(* CoDeSys 2.3 export: CANOPEN_UNIVERSAL_MASTER.EXP *)
(* Libraries: 05_Utilities\MPLCUtilities.lib 30.1.17 00:00:00, 11_System\SysLibFileAsync.lib 27.1.17 13:50:06, 11_System\SysLibRtc.lib 27.1.17 13:50:06, 12_Additional\Util.lib 27.1.17 13:50:06 *)

(* POU CodeSamples/CANopen/UniversalMaster/PRG_CANopen_IVO_AbsEncoder, FBD *)
(************************************************************************************
*
*                 Code sample  " PRG_CANopen_IVO_AbsEncoder "                 
*
*************************************************************************************
*
* (c) 2009 by SEW-EURODRIVE GmbH & Co KG
*
************************************************************************************
************************************************************************************
*
* PRG_CANopen_IVO_AbsEncoder
*
* This code sample demonstrates, how to configure and connect a 
* CANOpen IVO absolute encoder via CAN.
*
* Remarks : 
* - Use CANopen devices on a separate CAN and don´t mix it with SEW drives.
* - Set the Baudrate in plc configuration 
* 
************************************************************************************)
PROGRAM PRG_CANopen_IVO_AbsEncoder
VAR
	(* Configuration file IVO abs encoder *)
	fbConfig_IVO: FB_Configuration_CANopenSlave_IVO_AbsEncoder;
	stConfig_IVO: MC_EXTENDEDCONFIG_COSLAVE;
	bConfigDone_IVO: BOOL;

	(* Connect IVO abs encoder *)
	fbConnect_IVO: MPLC_ConnectUniversalSlave_CANopen;
	bReset_IVO: BOOL;
	stDiag_IVO: MC_DIAG_COSLAVE;
	aInputs_IVO: ARRAY [1..32] OF ARRAY [1..4] OF WORD;
	aOutputs_IVO: ARRAY [1..32] OF ARRAY [1..4] OF WORD;
	bConnectDone_IVO: BOOL;
	bConnectError_IVO: BOOL;
	nConnectErrorID_IVO: UDINT;
	stAxis_IVO: AXIS_REF;
END_VAR
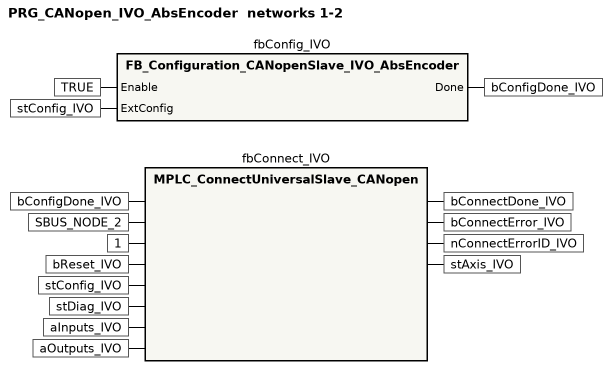
_FBD_ (* Function Block Diagram *)
NETWORK 1
	fbConfig_IVO:FB_Configuration_CANopenSlave_IVO_AbsEncoder(Enable: TRUE, ExtConfig: stConfig_IVO) => bConfigDone_IVO
NETWORK 2
	fbConnect_IVO:MPLC_ConnectUniversalSlave_CANopen(bConfigDone_IVO, SBUS_NODE_2, 1, bReset_IVO, stConfig_IVO, stDiag_IVO, aInputs_IVO, aOutputs_IVO, out 2 => bConnectError_IVO, out 3 => nConnectErrorID_IVO, out 4 => stAxis_IVO) => bConnectDone_IVO
_END_FBD_
(* the same logic as Structured Text *)
(* Network 1 *)
fbConfig_IVO(Enable := TRUE, ExtConfig := stConfig_IVO);
bConfigDone_IVO := fbConfig_IVO.Done;
(* Network 2: see the listing above *)
END_PROGRAM

(* POU CodeSamples/CANopen/UniversalMaster/FB_Configuration_CANopenSlave_IVO_AbsEncoder, ST *)
FUNCTION_BLOCK FB_Configuration_CANopenSlave_IVO_AbsEncoder
VAR_INPUT
	Enable: BOOL; 			(* Activate config *)
END_VAR
VAR_OUTPUT
	Done: BOOL;				(* Config done *)
END_VAR
VAR_IN_OUT
	ExtConfig : MC_EXTENDEDCONFIG_COSLAVE	;
	(*
		########################################################################################################
			MC_EXTENDEDCONFIG_COSLAVE
		#########################################################################################################

						
		Variable								Value			Description
		-------------------------------------------------------------------------------------------------------------------------------------------------------------
		bWaitBeforeOperational 				BOOL;			When TRUE, after the coupler has been parameterized, it won't be switched in operational
																before this variable is FALSE. This can be used for example, to store the configuration with the FB
																MPLC_Universal_CANopen, with Service "SEWIOS_STORE", after a reset of the coppler 
		-------------------------------------------------------------------------------------------------------------------------------------------------------------
		bNoSettingsDownload 				BOOL;			TRUE : No configuration of the module. The configuration has to be done manually.
		-------------------------------------------------------------------------------------------------------------------------------------------------------------
		bResetUnconditional 					BOOL;			Even if the Connect FB isn't in fault it is possible to reset the bus coppler
		-------------------------------------------------------------------------------------------------------------------------------------------------------------
		bIOHold 								BOOL;			TRUE : Input data remain unchanged and the output data are not resetet also if the FB is in fault 
		-------------------------------------------------------------------------------------------------------------------------------------------------------------
		TimeOutHeartBeat					UINT;			If this value (ms) is different to zero, HeartbeatMode will be activated
		-------------------------------------------------------------------------------------------------------------------------------------------------------------
		TimeOutNodeGuarding 				UINT;			If this value (ms) is different to zero, NodeGuarding will be activated. 
																Caution ! The MOVI-PLC basic doesn´t support NodeGuarding 
		-------------------------------------------------------------------------------------------------------------------------------------------------------------
		TimeOutInitSequence					UINT;			Timeout for initialisation sequence (seconds) 
		-------------------------------------------------------------------------------------------------------------------------------------------------------------
		NumberOfRxPDO 					UINT;			Receive PDO : MOVI-PLC --> Slave  max. 32 
		-------------------------------------------------------------------------------------------------------------------------------------------------------------
		NumberOfTxPDO 						UINT;			Send PDO :      Slave --> MOVI-PLC  max 32 
		-------------------------------------------------------------------------------------------------------------------------------------------------------------	
		SyncTime 								USINT;			Cycle time of the sync telegram in ms. 
																Default = 0 : no sync will be started.
																If  SyncTime > 0, this FB initializes a sync telegram with the ID set at SyncCOBID. 
																The slave has to support synchronous communication 
		-------------------------------------------------------------------------------------------------------------------------------------------------------------
		SyncCOBID							UINT;			Index 1005h. ID of the sync telegram. Usually 16#80. IF 0, the ID won't be written.
		-------------------------------------------------------------------------------------------------------------------------------------------------------------
		SyncTimeOut 							INT := -1;		Index 1006h. Normally equal to SyncTime. 
																The slave usually set SyncTimeOut equal to SyncTime * 1.5. 
																If < 0, the index won't be written. 0 means no control over the sync interval 
		-------------------------------------------------------------------------------------------------------------------------------------------------------------
		stInitialParameter_COSlave 			MC_INITIALPARAMETER_COSLAVE;
												(*#################################################################
												With this struct, user defined parameters will be written to the BusCoupler after the
												initialization of the MPLC_ConnectUniversalSlave_CANopen. 
												Add the following code to your program to initialise the struct : 
												Example:
												Index 16#6423:	Activates the event-driven transmission of PDOs with analog inputs
												Index 16#3500:	Index from the manufacturer specific profile area
	
													stInitialParameter_COSlave.aIndex[1] := 16#6423;  	(* Index to write to *)
													stInitialParameter_COSlave.aSubIndex[1] := 0;   	(* SubIndex to write to *)
													stInitialParameter_COSlave.aBytes[1] := 1;   		(* Number of bytes to write  *)
													stInitialParameter_COSlave.aData[1] := 1;   			(* Data *)
	
													stInitialParameter_COSlave.aIndex[2] := 16#3500;  	(* Index to write to *)
													stInitialParameter_COSlave.aSubIndex[2] := 0;   	(* SubIndex to write to *)
													stInitialParameter_COSlave.aBytes[2] := 2;   		(* Number of bytes to write *)
													stInitialParameter_COSlave.aData[2] := 5;   			(* Data *)
	
												If there are more than 10 (DHP11B) or 64 (DHx41B) parameters to write, declare 
												NUMOF_INITIALPARAMETER in your program.
	
													VAR_GLOBAL CONSTANT
														NUMOF_INITIALPARAMETER : UDINT := 20;	
													END_VAR
	
												##################################################################*)
			-------------------------------------------------------------------------------------------------------------------------------------------------------------
		(* IDs of the PDO telegrams. The IDs are always calculated with the following IDs as a basis + the address of the bus coupler *)

		RxPDO 								ARRAY[1..32] OF MC_PDO_COSLAVE;			(* MOVI-PLC --> Slave *)
												(* := 16#200,16#300,16#400,16#500,16#780,16#240,16#340,16#440,16#540,16#7C0;	*)
		-------------------------------------------------------------------------------------------------------------------------------------------------------------
		TxPDO 								ARRAY[1..32] OF MC_PDO_COSLAVE; 			(* Slave --> MOVI-PLC *)
												(*:= 16#180,16#280,16#380,16#480,16#680,16#1C0,16#2C0,16#3C0,16#4C0,16#6C0;*)
	*)
END_VAR
IF Enable AND NOT Done THEN

	(*########################################################

		Configuration of CANopenSlave (IVO AbsEncoder)
		
	#########################################################

		TransmissionType for TxPDOs and RxPDOs:

			0:										Event controlled and sychron (with SYNC-Object)
			1-240:									Cyclic and synchron (with SYNC-Object)
			254:									Producer specified
			255:									Acyclic and eventcontrolled 
			255 and EventTime = InhibitTime:	Cyclic

	#########################################################	*)


	(*************************************************** TxPDOs of CANOpenSlave ( MOVI-PLC ReceiveObjects) ***********************************************************)

	ExtConfig.NumberOfTxPDO				:= 1;		(*  TxPDO ---> CANopenSlave Transmit *)

	ExtConfig.TxPDO[1].EventTime			:= 20;		(* Slave: Index 0x18xx SubIndex 5: CycleTime in ms for CANopenSlave TXPDO *)
	ExtConfig.TxPDO[1].InhibitTime			:= 20;		(* Slave: Index 0x18xx SubIndex 3: InhibitTime in ms for CANopenSlave TxPDO *)
	ExtConfig.TxPDO[1].TransmissionType	:= 254;		(* Slave: Index 0x18xx SubIndex 2: TransmissionType for this TxPDO *)


	(*************************************************** RxPDOs of CANOpenSlave ( MOVI-PLC TransmitObjects) **********************************************************)

	ExtConfig.NumberOfRxPDO				:= 0;		(*  RxPDO ---> CANopenSlave Receive *)

	(* ExtConfig.RxPDO[1].EventTime		:= 0;		(* Master: CycleTime in ms for TransmitObjects (MOVI-PLC) *)
	ExtConfig.RxPDO[1].InhibitTime			:= 0;		(* Master: InhibitTime in ms for TransmitObjects (MOVI-PLC) *)
	ExtConfig.RxPDO[1].Length				:= 2;		(* Master: Length of this TransmitObject in bytes *)
	ExtConfig.RxPDO[1].TransmissionType	:= 255;		(* Slave: Index 0x14xx SubIndex 2: TransmissionType for this RxPDO *)*)


	(***************************************************** Additional parameters to set in the CANOpenSlave  ***************************************************************)

	(* Set rotation direction *)
	ExtConfig.stInitialParameter_COSlave.aIndex[1]			:= 16#6000;
	ExtConfig.stInitialParameter_COSlave.aSubIndex[1]	:= 0;
	ExtConfig.stInitialParameter_COSlave.aBytes[1]		:= 2;
	ExtConfig.stInitialParameter_COSlave.aData[1]			:= 0;		(* 0 = CV, 1 = CCV *)

	(* Write reference offset to AbsEncoder, Index 6003.0, data = new position *)
	(* Write Delivery state to AbsEncoder, Index 1011.1, data = 16#6C_6F_61_64 (load) *)
	(* Save values in Flash memory in the AbsEncoder, Index 1010.1, data = 16#73_61_76_65 (save) *)


	(********************************************** Additional configuration. Default values are in most cases sufficient *****************************************************)

	ExtConfig.bIOHold						:= FALSE;
	ExtConfig.bNoSettingsDownload			:= FALSE;
	ExtConfig.bWaitBeforeOperational		:= FALSE;
	ExtConfig.bResetUnconditional			:= FALSE;

	ExtConfig.TimeOutHeartBeat				:= 400;				(* [ms] *)
	ExtConfig.TimeOutNodeGuarding		:= 0;				(* [ms]. CAUTION ! DHP11B (MOVI-PLC basic) does NOT support NodeGuarding *)
	ExtConfig.TimeOutInitSequence			:= 5;				(* [seconds]. If the Init-Sequence takes longer than this TimeOut time --> Error *)
	ExtConfig.SyncCOBID						:= 0;				(* SyncObject ID for TransmissionType 0-240 (RxPDO). Usually 128. If 0, the ID will not be written *)
	ExtConfig.SyncTime						:= 0;				(* CycleTime for the SYNC-Object *)

	ExtConfig.TxPDO[1].COBID				:= 16#180;			(* In order to disable the use of RTR frames for the PDOs, set bit 30 = "RTR not allowed" *)
	ExtConfig.TxPDO[2].COBID				:= 16#280;			(* Ex. 16#4000_0280 *)
	ExtConfig.TxPDO[3].COBID				:= 16#380;
	ExtConfig.TxPDO[4].COBID				:= 16#480;			(* NOTE! These values are base values. The input "Address" will automatically be added *)
	ExtConfig.TxPDO[5].COBID				:= 16#680;
	ExtConfig.TxPDO[6].COBID				:= 16#1C0;
	ExtConfig.TxPDO[7].COBID				:= 16#2C0;
	ExtConfig.TxPDO[8].COBID				:= 16#3C0;
	ExtConfig.TxPDO[9].COBID				:= 16#4C0;
	ExtConfig.TxPDO[10].COBID				:= 16#6C0;

	ExtConfig.RxPDO[1].COBID				:= 16#200;
	ExtConfig.RxPDO[2].COBID				:= 16#300;
	ExtConfig.RxPDO[3].COBID				:= 16#400;
	ExtConfig.RxPDO[4].COBID				:= 16#500;
	ExtConfig.RxPDO[5].COBID				:= 16#780;
	ExtConfig.RxPDO[6].COBID				:= 16#240;
	ExtConfig.RxPDO[7].COBID				:= 16#340;
	ExtConfig.RxPDO[8].COBID				:= 16#440;
	ExtConfig.RxPDO[9].COBID				:= 16#540;
	ExtConfig.RxPDO[10].COBID				:= 16#7C0;

	Done := TRUE;

END_IF
END_FUNCTION_BLOCK

(* POU CodeSamples/CANopen/UniversalMaster/CANopen_activ, ST *)
(*######################################################
Functionblock:
- to send sync for the slave, to auto-detection of baudrate.
- set baudrate 
- set address 
#######################################################*)
FUNCTION_BLOCK CANopen_activ
VAR_INPUT
	Node: CAN_NODE; (* CAN_NODE_1 or CAN_NODE_2*)
	Address_Default : WORD;(* 0...127*)
	Address: WORD;			(* 1...63 *)
	Baudrate: WORD;(* 0 = 1 M , 2 = 500 k , 3 = 250 k baud*)
END_VAR
VAR_OUTPUT
	Done: BOOL; 				(* Connection to the CAN module successfully started *)
	Error: BOOL; 				(* Error within the function block *)
	ErrorID: UDINT; 			(* Error identification *)
END_VAR
VAR
	Init: BOOL;
	CanMsg: ST_CanAcyclicMsg;
	Timer: TON;
	l_State: UINT;
	StartAdresse_Diag: UINT;
	StartAdresse_Input: UINT;
	StartAdresse_Output: UINT;
	bMerkerCANSuspended: BOOL;
	SComCtrl1: SComControl;
	Counter: INT;
	fbSComCheckId: SComCheckId;
	SComRecSDO: SComReceive;
	SComRecNMT: SComReceive;
	SComRecEmergency: SComReceive;
	sSDORecDataTemp : sTwoDWORDData;
	NMT_Default_Byte : BYTE;
	NMT_Byte : BYTE;
	AbortCode: DWORD;
END_VAR
CASE l_State OF
(* ============ Initialisierung  Variablen =============== *)
	0:
		l_State := 10;

	10:
		IF ( Address < 1 ) OR ( Address > 63 ) OR (Address_Default > 127) THEN
			Error := TRUE;
			ErrorID := E_CAN_IO_MODULE_INVALID_PARAMETERS;
			RETURN;
		END_IF

		l_State := 50;

	50:
	(* SBus suspend --> damit können neue Objekte eingerichtet werden*)
      (* SCOM SUSPEND *)
	IF fTestAndSet( stInterlock.yTaskLock_CANSuspend ) THEN		(* CAN "belegen" damit keine andere Instanz Objekte anlegen will *)
		SEWMotionIntern.SComAllocationMax_I := SEWMotionIntern.SComAllocationMax_I - ( 12 + 4 * 2(*( xx.NbTxPDO + xx.NbCyclicRxPDO )*));
		SEWMotionIntern.SComAllocationMax_M := SEWMotionIntern.SComAllocationMax_M - ( 12 + 4 *2(* ( xx.NbTxPDO + xx.NbCyclicRxPDO )*));
		SEWMotionIntern.SComAllocationMax_Q := SEWMotionIntern.SComAllocationMax_Q - ( 12 + 4 * 2(*( xx.NbTxPDO + xx.NbCyclicRxPDO )*));
		StartAdresse_Diag := DWORD_TO_UINT (SEWMotionIntern.SComAllocationMax_M );
		StartAdresse_Input := DWORD_TO_UINT( SEWMotionIntern.SComAllocationMax_I );
		StartAdresse_Output := DWORD_TO_UINT( SEWMotionIntern.SComAllocationMax_Q );
		bMerkerCANSuspended := TRUE;
		SComCtrl1( Execute := FALSE );
		l_State := 60;
	END_IF

	60:
	(* SBus suspend --> damit können neue Objekte eingerichtet werden*)
      (* SCOM SUSPEND *)
	SComCtrl1(
		Execute := TRUE,
		Node := Node,
	 	Control := SCOM_CONTROL_SUSPEND,
		Error => Error,
		ErrorID => ErrorID );
       IF SComCtrl1.Done THEN
		l_State := 65;
	END_IF

	65:
	(* ID´s überprüfen für Adresse Default --> könnte durch andere SCOM Objekte schon belegt sein *)
	FOR Counter := 1 TO 6 DO
		IF (Counter = 6 )  THEN
			fbSComCheckId(
				Enable := TRUE,
				Node := Node,
				Id := 16#80);
		ELSE
			fbSComCheckId(
				Enable := TRUE,
				Node := Node,
				Id := ( Address_Default + aCOB_IDs_general_CO[Counter] ));
		END_IF
		IF fbSComCheckId.IsUsed OR NOT fbSComCheckId.Done OR ((Counter < 6 ) AND ( fbSComCheckId.Id = 16#80)) THEN
			Error := TRUE;
			ErrorID := E_CAN_IO_MODULE_CAN_ID_ERROR ;
			RETURN;
		ELSIF fbSComCheckId.Error THEN
			Error := TRUE;
			ErrorID := fbSComCheckId.ErrorID;
			RETURN;
		END_IF
	END_FOR
	l_State := 66;

	66:
	(* ID´s überprüfen für Adresse  --> könnte durch andere SCOM Objekte schon belegt sein *)
	FOR Counter := 1 TO 6 DO
		IF (Counter = 6 )  THEN
			fbSComCheckId(
				Enable := TRUE,
				Node := Node,
				Id := 16#80);
		ELSE
			fbSComCheckId(
				Enable := TRUE,
				Node := Node,
				Id := ( Address + aCOB_IDs_general_CO[Counter] ));
		END_IF
		IF fbSComCheckId.IsUsed OR NOT fbSComCheckId.Done OR ((Counter < 6 ) AND ( fbSComCheckId.Id = 16#80)) THEN
			Error := TRUE;
			ErrorID := E_CAN_IO_MODULE_CAN_ID_ERROR ;
			RETURN;
		ELSIF fbSComCheckId.Error THEN
			Error := TRUE;
			ErrorID := fbSComCheckId.ErrorID;
			RETURN;
		END_IF
	END_FOR
	SComRecSDO( Execute := FALSE );
	l_State := 70;

	70:
	(* Receive Objekt für Antwort Hochlauf Address_Default anlegen SDO*)
	SComRecSDO(
		Execute := TRUE,
		Node := Node,
		ID := 16#580 + Address_Default,
		Length := 8,
		DataDest := StartAdresse_Input,
		DiagDest := StartAdresse_Diag,
		Error => Error,
		ErrorID => ErrorID );
	IF SComRecSDO.Done THEN
		StartAdresse_Input := StartAdresse_Input + 4;
		StartAdresse_Diag := StartAdresse_Diag + 4;
		StartAdresse_Output := StartAdresse_Output + 4;
		SEWInternCOSlave[Address_Default].LibIn := SComRecSDO.DataDest;
		SComRecNMT( Execute := FALSE );
   		 l_State := 72;
	END_IF

	72:
	(* Receive Objekt für Antwort Hochlauf Address_Default anlegen NMT*)
	SComRecNMT(
		Execute := TRUE,
		Node := Node,
		ID := 16#700 + Address_Default,
		Length := 1,
		DataDest := StartAdresse_Input,
		DiagDest := StartAdresse_Diag,
		Error => Error,
		ErrorID => ErrorID );
	IF SComRecSDO.Done THEN
		StartAdresse_Input := StartAdresse_Input + 2;
		StartAdresse_Diag := StartAdresse_Diag + 2;
		StartAdresse_Output := StartAdresse_Output + 2;
		SComRecNMT( Execute := FALSE );
   		 l_State := 73;
	END_IF

	73:
	(* Receive Objekt für Antwort Hochlauf Address anlegen NMT*)
	SComRecNMT(
		Execute := TRUE,
		Node := Node,
		ID := 16#700 + Address,
		Length := 8,
		DataDest := StartAdresse_Input,
		DiagDest := StartAdresse_Diag,
		Error => Error,
		ErrorID => ErrorID );
	IF SComRecSDO.Done THEN
		StartAdresse_Input := StartAdresse_Input + 2;
		StartAdresse_Diag := StartAdresse_Diag + 2;
		StartAdresse_Output := StartAdresse_Output + 2;
		SComRecEmergency( Execute := FALSE );
   		 l_State := 74;
	END_IF

	74:
	(* Receive Objekt für Emergency Object einstellen *)
   	 SComRecEmergency(
		Execute := TRUE,
		Node := Node,
		ID := 16#80 + Address_Default,
		Length := 8,
		DataDest := StartAdresse_Input,
		DiagDest := StartAdresse_Diag,
		Error => Error,
		ErrorID => ErrorID);
	IF SComRecEmergency.Done THEN
		SComCtrl1( Execute := FALSE );
		l_State := 80;
	END_IF

	80:
	(* SBUS einschalten *)
	SComCtrl1(
		Execute := TRUE,
		Node := Node,
		Control := SCOM_CONTROL_ON );
	(* SBUS Initialisierung abgeschlossen *)
	IF SComCtrl1.Done THEN
		stInterlock.yTaskLock_CANSuspend := 0;
		bMerkerCANSuspended := FALSE;
		l_State := 90;
	END_IF

	90:
	(* Synch senden damit der Slave die Baudrate erkennt *)
		IF NOT Init THEN
			CanMsg := F_WriteCanMsg(
										Node := Node,
										ID := 16#80,
										Length := 1,
										Data1:= 0,
										Data2 := 0,
										Data3 := 0,
										Data4 := 0,
										SBUSGateway_LogAdr := 0 );
			IF ( CanMsg.State = GEN_1_BUFFSTATE_INSERTED ) THEN
				Init :=TRUE;
			END_IF
		ELSIF Init THEN
			CanMsg.Result :=F_ResultCanMsg(CanAcyclicMsg := CanMsg);
			IF ( CanMsg.Result = GEN_3_BUFFSTATE_COMPLETED_SUCCESSFUL ) THEN
				Init := FALSE;
				l_State := 92;
			(* Fehler beim Senden --> Nachricht ging verloren --> nochmals *)
			ELSIF (CanMsg.Result = GEN_5_BUFFSTATE_COMPLETED_MSG_LOST ) THEN
				Init := FALSE;
			(* Fehler beim Senden --> Non-recovery error from CAN --> nochmals *)
			ELSIF (CanMsg.Result = GEN_4_BUFFSTATE_COMPLETED_ERROR ) THEN
				Init := FALSE;
			END_IF
		END_IF

	92: (* Kontrolle ob Slave mit Address_Default antwortet *)
	Timer(	IN := TRUE, PT := t#1s );
	IF NOT Timer.Q THEN
		ConfDataEx_ReadFromIoBuffer( SEWInternCOSlave[Address_Default].LibIn+4, BUFSEL_IN, ADR(NMT_Default_Byte), 1);
		ConfDataEx_ReadFromIoBuffer( SEWInternCOSlave[Address_Default].LibIn+6, BUFSEL_IN, ADR(NMT_Byte), 1);
		IF NMT_Default_Byte = 0 THEN
			IF NMT_Byte = 0 THEN
				l_State := 90;
			ELSE
				l_State := 100;
			END_IF
		ELSE
			l_State := 100;
		END_IF
	ELSE
		l_State := 100;
	END_IF

	100:
	(* Baudrate einstellen *)
	Timer(	IN := TRUE, PT := t#100ms );
	IF Timer.Q THEN
		IF NOT Init THEN
			CanMsg := F_WriteCanMsg(
										Node := Node,
										ID := 16#600+Address_Default,
										Length := 8,
										Data1:= 16#2F00,
										Data2 := 16#2100,
										Data3 := SHL(Baudrate,8),
										Data4 := 0,
										SBUSGateway_LogAdr := 0 );
			IF ( CanMsg.State = GEN_1_BUFFSTATE_INSERTED ) THEN
				Init :=TRUE;
			END_IF
		ELSIF Init THEN
			CanMsg.Result :=F_ResultCanMsg(CanAcyclicMsg := CanMsg);
			IF ( CanMsg.Result = GEN_3_BUFFSTATE_COMPLETED_SUCCESSFUL ) THEN
				Init := FALSE;
				Timer( IN := FALSE );
				l_State := 110;
			(* Fehler beim Senden --> Nachricht ging verloren --> nochmals *)
			ELSIF (CanMsg.Result = GEN_5_BUFFSTATE_COMPLETED_MSG_LOST ) THEN
				Init := FALSE;
				Timer( IN := FALSE );
			(* Fehler beim Senden --> Non-recovery error from CAN --> nochmals *)
			ELSIF (CanMsg.Result = GEN_4_BUFFSTATE_COMPLETED_ERROR ) THEN
				Init := FALSE;
				Timer( IN := FALSE );
			END_IF
		END_IF
	END_IF

	110:
		ConfDataEx_ReadFromIoBuffer( SEWInternCOSlave[Address_Default].LibIn, BUFSEL_IN, ADR(sSDORecDataTemp), 8);
		IF MAX_NUMBER_AXIS <> 12 THEN
			sSDORecDataTemp.DWORD1 := fSwapUDINTtoIntel(sSDORecDataTemp.DWORD1);
			sSDORecDataTemp.DWORD2 := fSwapUDINTtoIntel(sSDORecDataTemp.DWORD2);
		END_IF
		IF (sSDORecDataTemp.DWORD1 AND 16#FFFF_FFF0) = (16#0021002F AND 16#FFFF_FF00) + 16#60 THEN
				l_State := 120;
		ELSIF sSDORecDataTemp.DWORD1= (16#0021002F AND 16#FFFF_FF00) + 16#80 THEN
			Error := TRUE;
			ErrorID := E_CAN_IO_MODULE_INVALID_PARAMETERS;			(* Parameter error *)
			AbortCode := sSDORecDataTemp.DWORD2;	(* SDO abort code *)
		ELSE
			(* Time out *)
			Timer( IN := TRUE, PT := T#500ms);
			IF Timer.Q THEN
				Error := TRUE;
				ErrorID := E_CAN_IO_MODULE_TIME_OUT_SBUS;			(* Parameter transfer Time out *)
			END_IF
		END_IF

	120:
	(* ID einstellen *)
	Timer(	IN := TRUE, PT := t#100ms );
	IF Timer.Q THEN
		IF NOT Init THEN
			CanMsg := F_WriteCanMsg(
										Node := Node,
										ID := 16#600+Address_Default,
										Length := 8,
										Data1:= 16#2F01,
										Data2 := 16#2100,
										Data3 := SHL(Address,8),
										Data4 := 0,
										SBUSGateway_LogAdr := 0 );
			IF ( CanMsg.State = GEN_1_BUFFSTATE_INSERTED ) THEN
				Init :=TRUE;
			END_IF
		ELSIF Init THEN
			CanMsg.Result :=F_ResultCanMsg(CanAcyclicMsg := CanMsg);
			IF ( CanMsg.Result = GEN_3_BUFFSTATE_COMPLETED_SUCCESSFUL ) THEN
				Init := FALSE;
				Timer( IN := FALSE );
				l_State := 130;
			(* Fehler beim Senden --> Nachricht ging verloren --> nochmals *)
			ELSIF (CanMsg.Result = GEN_5_BUFFSTATE_COMPLETED_MSG_LOST ) THEN
				Init := FALSE;
				Timer( IN := FALSE );
			(* Fehler beim Senden --> Non-recovery error from CAN --> nochmals *)
			ELSIF (CanMsg.Result = GEN_4_BUFFSTATE_COMPLETED_ERROR ) THEN
				Init := FALSE;
				Timer( IN := FALSE );
			END_IF
		END_IF
	END_IF

	130:
		ConfDataEx_ReadFromIoBuffer( SEWInternCOSlave[Address_Default].LibIn, BUFSEL_IN, ADR(sSDORecDataTemp), 8);
		IF MAX_NUMBER_AXIS <> 12 THEN
			sSDORecDataTemp.DWORD1 := fSwapUDINTtoIntel(sSDORecDataTemp.DWORD1);
			sSDORecDataTemp.DWORD2 := fSwapUDINTtoIntel(sSDORecDataTemp.DWORD2);
		END_IF
		IF (sSDORecDataTemp.DWORD1 AND 16#FFFF_FFF0) = (16#0021012F AND 16#FFFF_FF00) + 16#60 THEN
				l_State := 140;
		ELSIF sSDORecDataTemp.DWORD1= (16#0021012F AND 16#FFFF_FF00) + 16#80 THEN
			Error := TRUE;
			ErrorID := E_CAN_IO_MODULE_INVALID_PARAMETERS;			(* Parameter error *)
			AbortCode := sSDORecDataTemp.DWORD2;	(* SDO abort code *)
		ELSE
			(* Time out *)
			Timer( IN := TRUE, PT := T#500ms);
			IF Timer.Q THEN
				Error := TRUE;
				ErrorID := E_CAN_IO_MODULE_TIME_OUT_SBUS;			(* Parameter transfer Time out *)
			END_IF
		END_IF

	140:
	(* Parameter save *)
	Timer(	IN := TRUE, PT := t#100ms );
	IF Timer.Q THEN
		IF NOT Init THEN
			CanMsg := F_WriteCanMsg(
										Node := Node,
										ID := 16#600+Address_Default,
										Length := 8,
										Data1:= 16#2310,
										Data2 := 16#1001,
										Data3 := 16#7361,
										Data4 := 16#7665,
										SBUSGateway_LogAdr := 0 );
			IF ( CanMsg.State = GEN_1_BUFFSTATE_INSERTED ) THEN
				Init :=TRUE;
			END_IF
		ELSIF Init THEN
			CanMsg.Result :=F_ResultCanMsg(CanAcyclicMsg := CanMsg);
			IF ( CanMsg.Result = GEN_3_BUFFSTATE_COMPLETED_SUCCESSFUL ) THEN
				Init := FALSE;
				Timer( IN := FALSE );
				l_State := 150;
			(* Fehler beim Senden --> Nachricht ging verloren --> nochmals *)
			ELSIF (CanMsg.Result = GEN_5_BUFFSTATE_COMPLETED_MSG_LOST ) THEN
				Init := FALSE;
				Timer( IN := FALSE );
			(* Fehler beim Senden --> Non-recovery error from CAN --> nochmals *)
			ELSIF (CanMsg.Result = GEN_4_BUFFSTATE_COMPLETED_ERROR ) THEN
				Init := FALSE;
				Timer( IN := FALSE );
			END_IF
		END_IF
	END_IF

	150:
		ConfDataEx_ReadFromIoBuffer( SEWInternCOSlave[Address_Default].LibIn, BUFSEL_IN, ADR(sSDORecDataTemp), 8);
		IF MAX_NUMBER_AXIS <> 12 THEN
			sSDORecDataTemp.DWORD1 := fSwapUDINTtoIntel(sSDORecDataTemp.DWORD1);
			sSDORecDataTemp.DWORD2 := fSwapUDINTtoIntel(sSDORecDataTemp.DWORD2);
		END_IF
		IF (sSDORecDataTemp.DWORD1 AND 16#FFFF_FFF0) = (16#01101023 AND 16#FFFF_FF00) + 16#60 THEN
				l_State := 200;
		ELSIF sSDORecDataTemp.DWORD1= (16#01101023 AND 16#FFFF_FF00) + 16#80 THEN
			Error := TRUE;
			ErrorID := E_CAN_IO_MODULE_INVALID_PARAMETERS;			(* Parameter error *)
			AbortCode := sSDORecDataTemp.DWORD2;	(* SDO abort code *)
		ELSE
			(* Time out *)
			Timer( IN := TRUE, PT := T#500ms);
			IF Timer.Q THEN
				Error := TRUE;
				ErrorID := E_CAN_IO_MODULE_TIME_OUT_SBUS;			(* Parameter transfer Time out *)
			END_IF
		END_IF

	200:
		Done := TRUE;
		Error := FALSE;
		ErrorID := 0;

END_CASE
END_FUNCTION_BLOCK

(* POU CodeSamples/CANopen/UniversalMaster/FB_Configuration_CANopenSlave_Beckhoff_BK5120, ST *)
FUNCTION_BLOCK FB_Configuration_CANopenSlave_Beckhoff_BK5120
VAR_INPUT
	Enable: BOOL; 			(* Activate config *)
END_VAR
VAR_OUTPUT
	Done: BOOL;				(* Config done *)
END_VAR
VAR_IN_OUT
	ExtConfig : MC_EXTENDEDCONFIG_COSLAVE	;
	(*
		########################################################################################################
			MC_EXTENDEDCONFIG_COSLAVE
		#########################################################################################################

						
		Variable								Value			Description
		-------------------------------------------------------------------------------------------------------------------------------------------------------------
		bWaitBeforeOperational 				BOOL;			When TRUE, after the coupler has been parameterized, it won't be switched in operational
																before this variable is FALSE. This can be used for example, to store the configuration with the FB
																MPLC_Universal_CANopen, with Service "SEWIOS_STORE", after a reset of the coppler 
		-------------------------------------------------------------------------------------------------------------------------------------------------------------
		bNoSettingsDownload 				BOOL;			TRUE : No configuration of the module. The configuration has to be done manually.
		-------------------------------------------------------------------------------------------------------------------------------------------------------------
		bResetUnconditional 					BOOL;			Even if the Connect FB isn't in fault it is possible to reset the bus coppler
		-------------------------------------------------------------------------------------------------------------------------------------------------------------
		bIOHold 								BOOL;			TRUE : Input data remain unchanged and the output data are not resetet also if the FB is in fault 
		-------------------------------------------------------------------------------------------------------------------------------------------------------------
		TimeOutHeartBeat					UINT;			If this value (ms) is different to zero, HeartbeatMode will be activated
		-------------------------------------------------------------------------------------------------------------------------------------------------------------
		TimeOutNodeGuarding 				UINT;			If this value (ms) is different to zero, NodeGuarding will be activated. 
																Caution ! The MOVI-PLC basic doesn´t support NodeGuarding 
		-------------------------------------------------------------------------------------------------------------------------------------------------------------
		TimeOutInitSequence					UINT;			Timeout for initialisation sequence (seconds) 
		-------------------------------------------------------------------------------------------------------------------------------------------------------------
		NumberOfRxPDO 					UINT;			Receive PDO : MOVI-PLC --> Slave  max. 32 
		-------------------------------------------------------------------------------------------------------------------------------------------------------------
		NumberOfTxPDO 						UINT;			Send PDO :      Slave --> MOVI-PLC  max 32 
		-------------------------------------------------------------------------------------------------------------------------------------------------------------	
		SyncTime 								USINT;			Cycle time of the sync telegram in ms. 
																Default = 0 : no sync will be started.
																If  SyncTime > 0, this FB initializes a sync telegram with the ID set at SyncCOBID. 
																The slave has to support synchronous communication 
		-------------------------------------------------------------------------------------------------------------------------------------------------------------
		SyncCOBID							UINT;			Index 1005h. ID of the sync telegram. Usually 16#80. IF 0, the ID won't be written.
		-------------------------------------------------------------------------------------------------------------------------------------------------------------
		SyncTimeOut 							INT := -1;		Index 1006h. Normally equal to SyncTime. 
																The slave usually set SyncTimeOut equal to SyncTime * 1.5. 
																If < 0, the index won't be written. 0 means no control over the sync interval 
		-------------------------------------------------------------------------------------------------------------------------------------------------------------
		stInitialParameter_COSlave 			MC_INITIALPARAMETER_COSLAVE;
												(*#################################################################
												With this struct, user defined parameters will be written to the BusCoupler after the
												initialization of the MPLC_ConnectUniversalSlave_CANopen. 
												Add the following code to your program to initialise the struct : 
												Example:
												Index 16#6423:	Activates the event-driven transmission of PDOs with analog inputs
												Index 16#3500:	Index from the manufacturer specific profile area
	
													stInitialParameter_COSlave.aIndex[1] := 16#6423;  	(* Index to write to *)
													stInitialParameter_COSlave.aSubIndex[1] := 0;   	(* SubIndex to write to *)
													stInitialParameter_COSlave.aBytes[1] := 1;   		(* Number of bytes to write  *)
													stInitialParameter_COSlave.aData[1] := 1;   			(* Data *)
	
													stInitialParameter_COSlave.aIndex[2] := 16#3500;  	(* Index to write to *)
													stInitialParameter_COSlave.aSubIndex[2] := 0;   	(* SubIndex to write to *)
													stInitialParameter_COSlave.aBytes[2] := 2;   		(* Number of bytes to write *)
													stInitialParameter_COSlave.aData[2] := 5;   			(* Data *)
	
												If there are more than 10 (DHP11B) or 64 (DHx41B) parameters to write, declare 
												NUMOF_INITIALPARAMETER in your program.
	
													VAR_GLOBAL CONSTANT
														NUMOF_INITIALPARAMETER : UDINT := 20;	
													END_VAR
	
												##################################################################*)
			-------------------------------------------------------------------------------------------------------------------------------------------------------------
		(* IDs of the PDO telegrams. The IDs are always calculated with the following IDs as a basis + the address of the bus coupler *)

		RxPDO 								ARRAY[1..32] OF MC_PDO_COSLAVE;			(* MOVI-PLC --> Slave *)
												(* := 16#200,16#300,16#400,16#500,16#780,16#240,16#340,16#440,16#540,16#7C0;	*)
		-------------------------------------------------------------------------------------------------------------------------------------------------------------
		TxPDO 								ARRAY[1..32] OF MC_PDO_COSLAVE; 			(* Slave --> MOVI-PLC *)
												(*:= 16#180,16#280,16#380,16#480,16#680,16#1C0,16#2C0,16#3C0,16#4C0,16#6C0;*)
	*)
END_VAR
IF Enable AND NOT Done THEN

	(*########################################################

		Configuration of CANopenSlave (Beckhoff BK5120)
		
	#########################################################

		TransmissionType for TxPDOs and RxPDOs:

			0:										Event controlled and sychron (with SYNC-Object)
			1-240:									Cyclic and synchron (with SYNC-Object)
			254:									Producer specified
			255:									Acyclic and eventcontrolled 
			255 and EventTime = InhibitTime:	Cyclic

	#########################################################	*)


	(*************************************************** TxPDOs of CANOpenSlave ( MOVI-PLC ReceiveObjects) ***********************************************************)

	ExtConfig.NumberOfTxPDO				:= 2;		(*  TxPDO ---> CANopenSlave Transmit *)

	ExtConfig.TxPDO[1].EventTime			:= 200;		(* Slave: Index 0x18xx SubIndex 5: CycleTime in ms for CANopenSlave TXPDO *)
	ExtConfig.TxPDO[1].InhibitTime			:= 5;		(* Slave: Index 0x18xx SubIndex 3: InhibitTime in ms for CANopenSlave TxPDO *)
	ExtConfig.TxPDO[1].TransmissionType	:= 255;		(* Slave: Index 0x18xx SubIndex 2: TransmissionType for this TxPDO *)

	ExtConfig.TxPDO[2].EventTime			:= 100;		(* Slave: Index 0x18xx SubIndex 5: CycleTime in ms for CANopenSlave TXPDO *)
	ExtConfig.TxPDO[2].InhibitTime			:= 100;		(* Slave: Index 0x18xx SubIndex 3: InhibitTime in ms for CANopenSlave TxPDO *)
	ExtConfig.TxPDO[2].TransmissionType	:= 255;		(* Slave: Index 0x18xx SubIndex 2: TransmissionType for this TxPDO *)


	(*************************************************** RxPDOs of CANOpenSlave ( MOVI-PLC TransmitObjects) **********************************************************)

	ExtConfig.NumberOfRxPDO				:= 2;		(*  RxPDO ---> CANopenSlave Receive *)

	ExtConfig.RxPDO[1].EventTime			:= 200;		(* Master: CycleTime in ms for TransmitObjects (MOVI-PLC) *)
	ExtConfig.RxPDO[1].InhibitTime			:= 5;		(* Master: InhibitTime in ms for TransmitObjects (MOVI-PLC) *)
	ExtConfig.RxPDO[1].Length				:= 8;		(* Master: Length of this TransmitObject in bytes *)
	ExtConfig.RxPDO[1].TransmissionType	:= 255;		(* Slave: Index 0x14xx SubIndex 2: TransmissionType for this RxPDO *)

	ExtConfig.RxPDO[2].EventTime			:= 100;		(* Master: CycleTime in ms for TransmitObjects (MOVI-PLC) *)
	ExtConfig.RxPDO[2].InhibitTime			:= 100;		(* Master: InhibitTime in ms for TransmitObjects (MOVI-PLC) *)
	ExtConfig.RxPDO[2].Length				:= 8;		(* Master: Length of this TransmitObject in bytes *)
	ExtConfig.RxPDO[2].TransmissionType	:= 255;		(* Slave: Index 0x14xx SubIndex 2: TransmissionType for this RxPDO *)


	(***************************************************** Additional parameters to set in the CANOpenSlave  ***************************************************************)

	(* Enable transmission of analog inputs *)
	ExtConfig.stInitialParameter_COSlave.aIndex[1]			:= 16#6423;
	ExtConfig.stInitialParameter_COSlave.aSubIndex[1]	:= 0;
	ExtConfig.stInitialParameter_COSlave.aBytes[1]		:= 1;
	ExtConfig.stInitialParameter_COSlave.aData[1]			:= 1;

(*	(* Disable write protection, step 1 *)
	ExtConfig.stInitialParameter_COSlave.aIndex[2]			:= 16#4500;
	ExtConfig.stInitialParameter_COSlave.aSubIndex[2]	:= 0;
	ExtConfig.stInitialParameter_COSlave.aBytes[2]		:= 4;
	ExtConfig.stInitialParameter_COSlave.aData[2]			:= 16#E302_AFFE;

	(* Disable write protection, step 2 *)
	ExtConfig.stInitialParameter_COSlave.aIndex[3]			:= 16#4500;
	ExtConfig.stInitialParameter_COSlave.aSubIndex[3]	:= 0;
	ExtConfig.stInitialParameter_COSlave.aBytes[3]		:= 4;
	ExtConfig.stInitialParameter_COSlave.aData[3]			:= 16#E301_0001;

	(* Disable write protection, step 3 *)
	ExtConfig.stInitialParameter_COSlave.aIndex[4]			:= 16#4500;
	ExtConfig.stInitialParameter_COSlave.aSubIndex[4]	:= 0;
	ExtConfig.stInitialParameter_COSlave.aBytes[4]		:= 4;
	ExtConfig.stInitialParameter_COSlave.aData[4]			:= 16#E300_0101;
*)

	(********************************************** Additional configuration. Default values are in most cases sufficient *****************************************************)

	ExtConfig.bIOHold						:= FALSE;
	ExtConfig.bNoSettingsDownload			:= FALSE;
	ExtConfig.bWaitBeforeOperational		:= FALSE;
	ExtConfig.bResetUnconditional			:= FALSE;

	ExtConfig.TimeOutHeartBeat				:= 400;				(* [ms] *)
	ExtConfig.TimeOutNodeGuarding		:= 0;				(* [ms]. CAUTION ! DHP11B (MOVI-PLC basic) does NOT support NodeGuarding *)
	ExtConfig.TimeOutInitSequence			:= 10;				(* [seconds]. If the Init-Sequence takes longer than this TimeOut time --> Error *)
	ExtConfig.SyncCOBID						:= 0;				(* SyncObject ID for TransmissionType 0-240 (RxPDO). Usually 128. If 0, the ID will not be written *)
	ExtConfig.SyncTime						:= 0;				(* CycleTime for the SYNC-Object *)

	ExtConfig.TxPDO[1].COBID				:= 16#180;			(* In order to disable the use of RTR frames for the PDOs, set bit 30 = "RTR not allowed" *)
	ExtConfig.TxPDO[2].COBID				:= 16#280;			(* Ex. 16#4000_0280 *)
	ExtConfig.TxPDO[3].COBID				:= 16#380;
	ExtConfig.TxPDO[4].COBID				:= 16#480;			(* NOTE! These values are base values. The input "Address" will automatically be added *)
	ExtConfig.TxPDO[5].COBID				:= 16#680;
	ExtConfig.TxPDO[6].COBID				:= 16#1C0;
	ExtConfig.TxPDO[7].COBID				:= 16#2C0;
	ExtConfig.TxPDO[8].COBID				:= 16#3C0;
	ExtConfig.TxPDO[9].COBID				:= 16#4C0;
	ExtConfig.TxPDO[10].COBID				:= 16#6C0;

	ExtConfig.RxPDO[1].COBID				:= 16#200;
	ExtConfig.RxPDO[2].COBID				:= 16#300;
	ExtConfig.RxPDO[3].COBID				:= 16#400;
	ExtConfig.RxPDO[4].COBID				:= 16#500;
	ExtConfig.RxPDO[5].COBID				:= 16#780;
	ExtConfig.RxPDO[6].COBID				:= 16#240;
	ExtConfig.RxPDO[7].COBID				:= 16#340;
	ExtConfig.RxPDO[8].COBID				:= 16#440;
	ExtConfig.RxPDO[9].COBID				:= 16#540;
	ExtConfig.RxPDO[10].COBID				:= 16#7C0;

	Done := TRUE;

END_IF
END_FUNCTION_BLOCK

(* POU CodeSamples/CANopen/UniversalMaster/FB_Configuration_CANopenSlave_FESTO_CPX, ST *)
FUNCTION_BLOCK FB_Configuration_CANopenSlave_FESTO_CPX
VAR_INPUT
	Enable: BOOL; 			(* Activate config *)
END_VAR
VAR_OUTPUT
	Done: BOOL;				(* Config done *)
END_VAR
VAR_IN_OUT
	ExtConfig : MC_EXTENDEDCONFIG_COSLAVE	;
	(*
		########################################################################################################
			MC_EXTENDEDCONFIG_COSLAVE
		#########################################################################################################

						
		Variable								Value			Description
		-------------------------------------------------------------------------------------------------------------------------------------------------------------
		bWaitBeforeOperational 				BOOL;			When TRUE, after the coupler has been parameterized, it won't be switched in operational
																before this variable is FALSE. This can be used for example, to store the configuration with the FB
																MPLC_Universal_CANopen, with Service "SEWIOS_STORE", after a reset of the coppler 
		-------------------------------------------------------------------------------------------------------------------------------------------------------------
		bNoSettingsDownload 				BOOL;			TRUE : No configuration of the module. The configuration has to be done manually.
		-------------------------------------------------------------------------------------------------------------------------------------------------------------
		bResetUnconditional 					BOOL;			Even if the Connect FB isn't in fault it is possible to reset the bus coppler
		-------------------------------------------------------------------------------------------------------------------------------------------------------------
		bIOHold 								BOOL;			TRUE : Input data remain unchanged and the output data are not resetet also if the FB is in fault 
		-------------------------------------------------------------------------------------------------------------------------------------------------------------
		TimeOutHeartBeat					UINT;			If this value (ms) is different to zero, HeartbeatMode will be activated
		-------------------------------------------------------------------------------------------------------------------------------------------------------------
		TimeOutNodeGuarding 				UINT;			If this value (ms) is different to zero, NodeGuarding will be activated. 
																Caution ! The MOVI-PLC basic doesn´t support NodeGuarding 
		-------------------------------------------------------------------------------------------------------------------------------------------------------------
		TimeOutInitSequence					UINT;			Timeout for initialisation sequence (seconds) 
		-------------------------------------------------------------------------------------------------------------------------------------------------------------
		NumberOfRxPDO 					UINT;			Receive PDO : MOVI-PLC --> Slave  max. 32 
		-------------------------------------------------------------------------------------------------------------------------------------------------------------
		NumberOfTxPDO 						UINT;			Send PDO :      Slave --> MOVI-PLC  max 32 
		-------------------------------------------------------------------------------------------------------------------------------------------------------------	
		SyncTime 								USINT;			Cycle time of the sync telegram in ms. 
																Default = 0 : no sync will be started.
																If  SyncTime > 0, this FB initializes a sync telegram with the ID set at SyncCOBID. 
																The slave has to support synchronous communication 
		-------------------------------------------------------------------------------------------------------------------------------------------------------------
		SyncCOBID							UINT;			Index 1005h. ID of the sync telegram. Usually 16#80. IF 0, the ID won't be written.
		-------------------------------------------------------------------------------------------------------------------------------------------------------------
		SyncTimeOut 							INT := -1;		Index 1006h. Normally equal to SyncTime. 
																The slave usually set SyncTimeOut equal to SyncTime * 1.5. 
																If < 0, the index won't be written. 0 means no control over the sync interval 
		-------------------------------------------------------------------------------------------------------------------------------------------------------------
		stInitialParameter_COSlave 			MC_INITIALPARAMETER_COSLAVE;
												(*#################################################################
												With this struct, user defined parameters will be written to the BusCoupler after the
												initialization of the MPLC_ConnectUniversalSlave_CANopen. 
												Add the following code to your program to initialise the struct : 
												Example:
												Index 16#6423:	Activates the event-driven transmission of PDOs with analog inputs
												Index 16#3500:	Index from the manufacturer specific profile area
	
													stInitialParameter_COSlave.aIndex[1] := 16#6423;  	(* Index to write to *)
													stInitialParameter_COSlave.aSubIndex[1] := 0;   	(* SubIndex to write to *)
													stInitialParameter_COSlave.aBytes[1] := 1;   		(* Number of bytes to write  *)
													stInitialParameter_COSlave.aData[1] := 1;   			(* Data *)
	
													stInitialParameter_COSlave.aIndex[2] := 16#3500;  	(* Index to write to *)
													stInitialParameter_COSlave.aSubIndex[2] := 0;   	(* SubIndex to write to *)
													stInitialParameter_COSlave.aBytes[2] := 2;   		(* Number of bytes to write *)
													stInitialParameter_COSlave.aData[2] := 5;   			(* Data *)
	
												If there are more than 10 (DHP11B) or 64 (DHx41B) parameters to write, declare 
												NUMOF_INITIALPARAMETER in your program.
	
													VAR_GLOBAL CONSTANT
														NUMOF_INITIALPARAMETER : UDINT := 20;	
													END_VAR
	
												##################################################################*)
			-------------------------------------------------------------------------------------------------------------------------------------------------------------
		(* IDs of the PDO telegrams. The IDs are always calculated with the following IDs as a basis + the address of the bus coupler *)

		RxPDO 								ARRAY[1..32] OF MC_PDO_COSLAVE;			(* MOVI-PLC --> Slave *)
												(* := 16#200,16#300,16#400,16#500,16#780,16#240,16#340,16#440,16#540,16#7C0;	*)
		-------------------------------------------------------------------------------------------------------------------------------------------------------------
		TxPDO 								ARRAY[1..32] OF MC_PDO_COSLAVE; 			(* Slave --> MOVI-PLC *)
												(*:= 16#180,16#280,16#380,16#480,16#680,16#1C0,16#2C0,16#3C0,16#4C0,16#6C0;*)
	*)
END_VAR
IF Enable AND NOT Done THEN

	(*########################################################

		Configuration of CANopenSlave FESTO CPX FB14
		
	#########################################################

		TransmissionType for TxPDOs and RxPDOs:

			0:										Event controlled and sychron (with SYNC-Object)
			1-240:									Cyclic and synchron (with SYNC-Object)
			254:									Producer specified
			255:									Acyclic and eventcontrolled 
			255 and EventTime = InhibitTime:	Cyclic

	#########################################################	*)


	(*************************************************** TxPDOs of CANOpenSlave ( MOVI-PLC ReceiveObjects) ***********************************************************)

	ExtConfig.NumberOfTxPDO				:= 4;		(*  TxPDO ---> CANopenSlave Transmit *)

	ExtConfig.TxPDO[1].EventTime			:= 200;		(* Slave: Index 0x18xx SubIndex 5: CycleTime in ms for CANopenSlave TXPDO *)
	ExtConfig.TxPDO[1].InhibitTime			:= 5;		(* Slave: Index 0x18xx SubIndex 3: InhibitTime in ms for CANopenSlave TxPDO *)
	ExtConfig.TxPDO[1].TransmissionType	:= 255;		(* Slave: Index 0x18xx SubIndex 2: TransmissionType for this TxPDO *)

	ExtConfig.TxPDO[2].EventTime			:= 100;		(* Slave: Index 0x18xx SubIndex 5: CycleTime in ms for CANopenSlave TXPDO *)
	ExtConfig.TxPDO[2].InhibitTime			:= 100;		(* Slave: Index 0x18xx SubIndex 3: InhibitTime in ms for CANopenSlave TxPDO *)
	ExtConfig.TxPDO[2].TransmissionType	:= 255;		(* Slave: Index 0x18xx SubIndex 2: TransmissionType for this TxPDO *)

	ExtConfig.TxPDO[3].EventTime			:= 100;		(* Slave: Index 0x18xx SubIndex 5: CycleTime in ms for CANopenSlave TXPDO *)
	ExtConfig.TxPDO[3].InhibitTime			:= 100;		(* Slave: Index 0x18xx SubIndex 3: InhibitTime in ms for CANopenSlave TxPDO *)
	ExtConfig.TxPDO[3].TransmissionType	:= 255;		(* Slave: Index 0x18xx SubIndex 2: TransmissionType for this TxPDO *)

	ExtConfig.TxPDO[4].EventTime			:= 100;		(* Slave: Index 0x18xx SubIndex 5: CycleTime in ms for CANopenSlave TXPDO *)
	ExtConfig.TxPDO[4].InhibitTime			:= 100;		(* Slave: Index 0x18xx SubIndex 3: InhibitTime in ms for CANopenSlave TxPDO *)
	ExtConfig.TxPDO[4].TransmissionType	:= 255;		(* Slave: Index 0x18xx SubIndex 2: TransmissionType for this TxPDO *)


	(*************************************************** RxPDOs of CANOpenSlave ( MOVI-PLC TransmitObjects) **********************************************************)

	ExtConfig.NumberOfRxPDO				:= 4;		(*  RxPDO ---> CANopenSlave Receive *)

	ExtConfig.RxPDO[1].EventTime			:= 200;		(* Master: CycleTime in ms for TransmitObjects (MOVI-PLC) *)
	ExtConfig.RxPDO[1].InhibitTime			:= 5;		(* Master: InhibitTime in ms for TransmitObjects (MOVI-PLC) *)
	ExtConfig.RxPDO[1].Length				:= 8;		(* Master: Length of this TransmitObject in bytes *)
	ExtConfig.RxPDO[1].TransmissionType	:= 255;		(* Slave: Index 0x14xx SubIndex 2: TransmissionType for this RxPDO *)

	ExtConfig.RxPDO[2].EventTime			:= 100;		(* Master: CycleTime in ms for TransmitObjects (MOVI-PLC) *)
	ExtConfig.RxPDO[2].InhibitTime			:= 100;		(* Master: InhibitTime in ms for TransmitObjects (MOVI-PLC) *)
	ExtConfig.RxPDO[2].Length				:= 8;		(* Master: Length of this TransmitObject in bytes *)
	ExtConfig.RxPDO[2].TransmissionType	:= 255;		(* Slave: Index 0x14xx SubIndex 2: TransmissionType for this RxPDO *)

	ExtConfig.RxPDO[3].EventTime			:= 100;		(* Master: CycleTime in ms for TransmitObjects (MOVI-PLC) *)
	ExtConfig.RxPDO[3].InhibitTime			:= 100;		(* Master: InhibitTime in ms for TransmitObjects (MOVI-PLC) *)
	ExtConfig.RxPDO[3].Length				:= 8;		(* Master: Length of this TransmitObject in bytes *)
	ExtConfig.RxPDO[3].TransmissionType	:= 255;		(* Slave: Index 0x14xx SubIndex 2: TransmissionType for this RxPDO *)

	ExtConfig.RxPDO[4].EventTime			:= 100;		(* Master: CycleTime in ms for TransmitObjects (MOVI-PLC) *)
	ExtConfig.RxPDO[4].InhibitTime			:= 100;		(* Master: InhibitTime in ms for TransmitObjects (MOVI-PLC) *)
	ExtConfig.RxPDO[4].Length				:= 8;		(* Master: Length of this TransmitObject in bytes *)
	ExtConfig.RxPDO[4].TransmissionType	:= 255;		(* Slave: Index 0x14xx SubIndex 2: TransmissionType for this RxPDO *)


	(***************************************************** Additional parameters to set in the CANOpenSlave  ***************************************************************)

(*	(* Enable transmission of analog inputs *)
	ExtConfig.stInitialParameter_COSlave.aIndex[1]			:= 16#6423;
	ExtConfig.stInitialParameter_COSlave.aSubIndex[1]	:= 0;
	ExtConfig.stInitialParameter_COSlave.aBytes[1]		:= 1;
	ExtConfig.stInitialParameter_COSlave.aData[1]			:= 1;
*)

	(********************************************** Additional configuration. Default values are in most cases sufficient *****************************************************)

	ExtConfig.bIOHold						:= FALSE;
	ExtConfig.bNoSettingsDownload			:= FALSE;
	ExtConfig.bWaitBeforeOperational		:= FALSE;
	ExtConfig.bResetUnconditional			:= FALSE;

	ExtConfig.TimeOutHeartBeat				:= 400;				(* [ms] *)
	ExtConfig.TimeOutNodeGuarding		:= 0;				(* [ms]. CAUTION ! DHP11B (MOVI-PLC basic) does NOT support NodeGuarding *)
	ExtConfig.TimeOutInitSequence			:= 10;				(* [seconds]. If the Init-Sequence takes longer than this TimeOut time --> Error *)
	ExtConfig.SyncCOBID						:= 0;				(* SyncObject ID for TransmissionType 0-240 (RxPDO). Usually 128. If 0, the ID will not be written *)
	ExtConfig.SyncTime						:= 0;				(* CycleTime for the SYNC-Object *)

	ExtConfig.TxPDO[1].COBID				:= 16#180;			(* In order to disable the use of RTR frames for the PDOs, set bit 30 = "RTR not allowed" *)
	ExtConfig.TxPDO[2].COBID				:= 16#280;			(* Ex. 16#4000_0280 *)
	ExtConfig.TxPDO[3].COBID				:= 16#380;
	ExtConfig.TxPDO[4].COBID				:= 16#480;			(* NOTE! These values are base values. The input "Address" will automatically be added *)
	ExtConfig.TxPDO[5].COBID				:= 16#680;
	ExtConfig.TxPDO[6].COBID				:= 16#1C0;
	ExtConfig.TxPDO[7].COBID				:= 16#2C0;
	ExtConfig.TxPDO[8].COBID				:= 16#3C0;
	ExtConfig.TxPDO[9].COBID				:= 16#4C0;
	ExtConfig.TxPDO[10].COBID				:= 16#6C0;

	ExtConfig.RxPDO[1].COBID				:= 16#200;
	ExtConfig.RxPDO[2].COBID				:= 16#300;
	ExtConfig.RxPDO[3].COBID				:= 16#400;
	ExtConfig.RxPDO[4].COBID				:= 16#500;
	ExtConfig.RxPDO[5].COBID				:= 16#780;
	ExtConfig.RxPDO[6].COBID				:= 16#240;
	ExtConfig.RxPDO[7].COBID				:= 16#340;
	ExtConfig.RxPDO[8].COBID				:= 16#440;
	ExtConfig.RxPDO[9].COBID				:= 16#540;
	ExtConfig.RxPDO[10].COBID				:= 16#7C0;

	Done := TRUE;

END_IF
END_FUNCTION_BLOCK

(* POU CodeSamples/CANopen/UniversalMaster/FB_Configuration_CANopenSlave_FRABA_AbsEncoder, ST *)
FUNCTION_BLOCK FB_Configuration_CANopenSlave_FRABA_AbsEncoder
VAR_INPUT
	Enable: BOOL; 			(* Activate config *)
END_VAR
VAR_OUTPUT
	Done: BOOL;				(* Config done *)
END_VAR
VAR_IN_OUT
	ExtConfig : MC_EXTENDEDCONFIG_COSLAVE	;
	(*
		########################################################################################################
			MC_EXTENDEDCONFIG_COSLAVE
		#########################################################################################################

						
		Variable								Value			Description
		-------------------------------------------------------------------------------------------------------------------------------------------------------------
		bWaitBeforeOperational 				BOOL;			When TRUE, after the coupler has been parameterized, it won't be switched in operational
																before this variable is FALSE. This can be used for example, to store the configuration with the FB
																MPLC_Universal_CANopen, with Service "SEWIOS_STORE", after a reset of the coppler 
		-------------------------------------------------------------------------------------------------------------------------------------------------------------
		bNoSettingsDownload 				BOOL;			TRUE : No configuration of the module. The configuration has to be done manually.
		-------------------------------------------------------------------------------------------------------------------------------------------------------------
		bResetUnconditional 					BOOL;			Even if the Connect FB isn't in fault it is possible to reset the bus coppler
		-------------------------------------------------------------------------------------------------------------------------------------------------------------
		bIOHold 								BOOL;			TRUE : Input data remain unchanged and the output data are not resetet also if the FB is in fault 
		-------------------------------------------------------------------------------------------------------------------------------------------------------------
		TimeOutHeartBeat					UINT;			If this value (ms) is different to zero, HeartbeatMode will be activated
		-------------------------------------------------------------------------------------------------------------------------------------------------------------
		TimeOutNodeGuarding 				UINT;			If this value (ms) is different to zero, NodeGuarding will be activated. 
																Caution ! The MOVI-PLC basic doesn´t support NodeGuarding 
		-------------------------------------------------------------------------------------------------------------------------------------------------------------
		TimeOutInitSequence					UINT;			Timeout for initialisation sequence (seconds) 
		-------------------------------------------------------------------------------------------------------------------------------------------------------------
		NumberOfRxPDO 					UINT;			Receive PDO : MOVI-PLC --> Slave  max. 32 
		-------------------------------------------------------------------------------------------------------------------------------------------------------------
		NumberOfTxPDO 						UINT;			Send PDO :      Slave --> MOVI-PLC  max 32 
		-------------------------------------------------------------------------------------------------------------------------------------------------------------	
		SyncTime 								USINT;			Cycle time of the sync telegram in ms. 
																Default = 0 : no sync will be started.
																If  SyncTime > 0, this FB initializes a sync telegram with the ID set at SyncCOBID. 
																The slave has to support synchronous communication 
		-------------------------------------------------------------------------------------------------------------------------------------------------------------
		SyncCOBID							UINT;			Index 1005h. ID of the sync telegram. Usually 16#80. IF 0, the ID won't be written.
		-------------------------------------------------------------------------------------------------------------------------------------------------------------
		SyncTimeOut 							INT := -1;		Index 1006h. Normally equal to SyncTime. 
																The slave usually set SyncTimeOut equal to SyncTime * 1.5. 
																If < 0, the index won't be written. 0 means no control over the sync interval 
		-------------------------------------------------------------------------------------------------------------------------------------------------------------
		stInitialParameter_COSlave 			MC_INITIALPARAMETER_COSLAVE;
												(*#################################################################
												With this struct, user defined parameters will be written to the BusCoupler after the
												initialization of the MPLC_ConnectUniversalSlave_CANopen. 
												Add the following code to your program to initialise the struct : 
												Example:
												Index 16#6423:	Activates the event-driven transmission of PDOs with analog inputs
												Index 16#3500:	Index from the manufacturer specific profile area
	
													stInitialParameter_COSlave.aIndex[1] := 16#6423;  	(* Index to write to *)
													stInitialParameter_COSlave.aSubIndex[1] := 0;   	(* SubIndex to write to *)
													stInitialParameter_COSlave.aBytes[1] := 1;   		(* Number of bytes to write  *)
													stInitialParameter_COSlave.aData[1] := 1;   			(* Data *)
	
													stInitialParameter_COSlave.aIndex[2] := 16#3500;  	(* Index to write to *)
													stInitialParameter_COSlave.aSubIndex[2] := 0;   	(* SubIndex to write to *)
													stInitialParameter_COSlave.aBytes[2] := 2;   		(* Number of bytes to write *)
													stInitialParameter_COSlave.aData[2] := 5;   			(* Data *)
	
												If there are more than 10 (DHP11B) or 64 (DHx41B) parameters to write, declare 
												NUMOF_INITIALPARAMETER in your program.
	
													VAR_GLOBAL CONSTANT
														NUMOF_INITIALPARAMETER : UDINT := 20;	
													END_VAR
	
												##################################################################*)
			-------------------------------------------------------------------------------------------------------------------------------------------------------------
		(* IDs of the PDO telegrams. The IDs are always calculated with the following IDs as a basis + the address of the bus coupler *)

		RxPDO 								ARRAY[1..32] OF MC_PDO_COSLAVE;			(* MOVI-PLC --> Slave *)
												(* := 16#200,16#300,16#400,16#500,16#780,16#240,16#340,16#440,16#540,16#7C0;	*)
		-------------------------------------------------------------------------------------------------------------------------------------------------------------
		TxPDO 								ARRAY[1..32] OF MC_PDO_COSLAVE; 			(* Slave --> MOVI-PLC *)
												(*:= 16#180,16#280,16#380,16#480,16#680,16#1C0,16#2C0,16#3C0,16#4C0,16#6C0;*)
	*)
END_VAR
IF Enable AND NOT Done THEN

	(*########################################################

		Configuration of CANopenSlave (FRABA AbsEncoder)
		
		NOTE! 
		The FRABA AbsEncoder occupy the chosen CAN address plus 1 on the
		CAN bus. Example: Switch inside the Absolute encoder is set to 9. The IDs
		used for CAN bus communication will correspond to adress 10.
		IMPORTANT! Set the address switch to one address lower than you intend
		to use. This way it will work well together with other CANopen modules on 
		the same bus, i.e. I/O modules etc.

			Wanted address:			10
			Abs.Enc. switch setting:	  9
			Input to function block:	10

	#########################################################

		TransmissionType for TxPDOs and RxPDOs:

			0:										Event controlled and sychron (with SYNC-Object)
			1-240:									Cyclic and synchron (with SYNC-Object)
			254:									Producer specified
			255:									Acyclic and eventcontrolled 
			255 and EventTime = InhibitTime:	Cyclic

	#########################################################	*)


	(*************************************************** TxPDOs of CANOpenSlave ( MOVI-PLC ReceiveObjects) ***********************************************************)

	ExtConfig.NumberOfTxPDO				:= 1;		(*  TxPDO ---> CANopenSlave Transmit *)

	ExtConfig.TxPDO[1].EventTime			:= 20;		(* Slave: Index 0x18xx SubIndex 5: CycleTime in ms for CANopenSlave TXPDO *)
	ExtConfig.TxPDO[1].InhibitTime			:= 20;		(* Slave: Index 0x18xx SubIndex 3: InhibitTime in ms for CANopenSlave TxPDO *)
	ExtConfig.TxPDO[1].TransmissionType	:= 255;		(* Slave: Index 0x18xx SubIndex 2: TransmissionType for this TxPDO *)


	(*************************************************** RxPDOs of CANOpenSlave ( MOVI-PLC TransmitObjects) **********************************************************)

	ExtConfig.NumberOfRxPDO				:= 0;		(*  RxPDO ---> CANopenSlave Receive *)

	(* ExtConfig.RxPDO[1].EventTime		:= 0;		(* Master: CycleTime in ms for TransmitObjects (MOVI-PLC) *)
	ExtConfig.RxPDO[1].InhibitTime			:= 0;		(* Master: InhibitTime in ms for TransmitObjects (MOVI-PLC) *)
	ExtConfig.RxPDO[1].Length				:= 2;		(* Master: Length of this TransmitObject in bytes *)
	ExtConfig.RxPDO[1].TransmissionType	:= 255;		(* Slave: Index 0x14xx SubIndex 2: TransmissionType for this RxPDO *)*)


	(***************************************************** Additional parameters to set in the CANOpenSlave  ***************************************************************)

	(* Set rotation direction *)
	ExtConfig.stInitialParameter_COSlave.aIndex[1]			:= 16#6000;
	ExtConfig.stInitialParameter_COSlave.aSubIndex[1]	:= 0;
	ExtConfig.stInitialParameter_COSlave.aBytes[1]		:= 2;
	ExtConfig.stInitialParameter_COSlave.aData[1]			:= 0;			(* 0 = CV, 1 = CCV *)

	(* Write reference offset to AbsEncoder, Index 2103.0, data = new position *)
	(* Save values in Flash memory in the AbsEncoder, Index 1010.1, data = 16#65766173 (evas) *)
	(* Write Delivery state to AbsEncoder, Index 1011.1, data = 16#64616F6C (daol) *)


	(********************************************** Additional configuration. Default values are in most cases sufficient *****************************************************)

	ExtConfig.bIOHold						:= FALSE;
	ExtConfig.bNoSettingsDownload			:= FALSE;
	ExtConfig.bWaitBeforeOperational		:= FALSE;
	ExtConfig.bResetUnconditional			:= FALSE;

	ExtConfig.bNoHeartBeat_Consumer			:= TRUE;
	ExtConfig.TimeOutHeartBeat				:= 400;				(* [ms] *)
	ExtConfig.TimeOutNodeGuarding		:= 0;				(* [ms]. CAUTION ! DHP11B (MOVI-PLC basic) does NOT support NodeGuarding *)
	ExtConfig.TimeOutInitSequence			:= 16;				(* [seconds]. If the Init-Sequence takes longer than this TimeOut time --> Error *)
	ExtConfig.SyncCOBID						:= 0;				(* SyncObject ID for TransmissionType 0-240 (RxPDO). Usually 128. If 0, the ID will not be written *)
	ExtConfig.SyncTime						:= 0;				(* CycleTime for the SYNC-Object *)

	ExtConfig.SBUSGateway_Address			:= 0(*1001*);			(* OSC71B Address,when used *)

	ExtConfig.TxPDO[1].COBID				:= 16#180;			(* In order to disable the use of RTR frames for the PDOs, set bit 30 = "RTR not allowed" *)
	ExtConfig.TxPDO[2].COBID				:= 16#280;			(* Ex. 16#4000_0280 *)
	ExtConfig.TxPDO[3].COBID				:= 16#380;
	ExtConfig.TxPDO[4].COBID				:= 16#480;			(* NOTE! These values are base values. The input "Address" will automatically be added *)
	ExtConfig.TxPDO[5].COBID				:= 16#680;
	ExtConfig.TxPDO[6].COBID				:= 16#1C0;
	ExtConfig.TxPDO[7].COBID				:= 16#2C0;
	ExtConfig.TxPDO[8].COBID				:= 16#3C0;
	ExtConfig.TxPDO[9].COBID				:= 16#4C0;
	ExtConfig.TxPDO[10].COBID				:= 16#6C0;

	ExtConfig.RxPDO[1].COBID				:= 16#200;
	ExtConfig.RxPDO[2].COBID				:= 16#300;
	ExtConfig.RxPDO[3].COBID				:= 16#400;
	ExtConfig.RxPDO[4].COBID				:= 16#500;
	ExtConfig.RxPDO[5].COBID				:= 16#780;
	ExtConfig.RxPDO[6].COBID				:= 16#240;
	ExtConfig.RxPDO[7].COBID				:= 16#340;
	ExtConfig.RxPDO[8].COBID				:= 16#440;
	ExtConfig.RxPDO[9].COBID				:= 16#540;
	ExtConfig.RxPDO[10].COBID				:= 16#7C0;

	Done := TRUE;

END_IF
END_FUNCTION_BLOCK

(* POU CodeSamples/CANopen/UniversalMaster/FB_Configuration_CANopenSlave_HBM, ST *)
FUNCTION_BLOCK FB_Configuration_CANopenSlave_HBM
(*Configuration for scalemodule HBM AD103C*)
VAR_INPUT
	Enable: BOOL; 			(* Activate config *)
END_VAR
VAR_OUTPUT
	Done: BOOL;				(* Config done *)
END_VAR
VAR_IN_OUT
	ExtConfig : MC_EXTENDEDCONFIG_COSLAVE	;
	(*
		########################################################################################################
			MC_EXTENDEDCONFIG_COSLAVE
		#########################################################################################################

						
		Variable								Value			Description
		-------------------------------------------------------------------------------------------------------------------------------------------------------------
		bWaitBeforeOperational 				BOOL;			When TRUE, after the coupler has been parameterized, it won't be switched in operational
																before this variable is FALSE. This can be used for example, to store the configuration with the FB
																MPLC_Universal_CANopen, with Service "SEWIOS_STORE", after a reset of the coppler 
		-------------------------------------------------------------------------------------------------------------------------------------------------------------
		bNoSettingsDownload 				BOOL;			TRUE : No configuration of the module. The configuration has to be done manually.
		-------------------------------------------------------------------------------------------------------------------------------------------------------------
		bResetUnconditional 					BOOL;			Even if the Connect FB isn't in fault it is possible to reset the bus coppler
		-------------------------------------------------------------------------------------------------------------------------------------------------------------
		bIOHold 								BOOL;			TRUE : Input data remain unchanged and the output data are not resetet also if the FB is in fault 
		-------------------------------------------------------------------------------------------------------------------------------------------------------------
		TimeOutHeartBeat					UINT;			If this value (ms) is different to zero, HeartbeatMode will be activated

		bNoHeartBeat_Producer:				BOOL := FALSE; (*Index 1017 SubIndex 0 not available *)
		-------------------------------------------------------------------------------------------------------------------------------------------------------------
		TimeOutNodeGuarding 				UINT;			If this value (ms) is different to zero, NodeGuarding will be activated. 
																Caution ! The MOVI-PLC basic doesn´t support NodeGuarding 
	
		bNoNodeGuarding:					BOOL:=FALSE; (* the Index of NodeGuarding isn`t available *)
		-------------------------------------------------------------------------------------------------------------------------------------------------------------
		TimeOutInitSequence					UINT;			Timeout for initialisation sequence (seconds) 
		-------------------------------------------------------------------------------------------------------------------------------------------------------------
		NumberOfRxPDO 					UINT;			Receive PDO : MOVI-PLC --> Slave  max. 32 
		-------------------------------------------------------------------------------------------------------------------------------------------------------------
		NumberOfTxPDO 						UINT;			Send PDO :      Slave --> MOVI-PLC  max 32 
		-------------------------------------------------------------------------------------------------------------------------------------------------------------	
		OffsetOfRxPDO:						UINT;			Offset for the 1. RxPDO
		-------------------------------------------------------------------------------------------------------------------------------------------------------------		
		OffsetOfTxPDO:						UINT;			Offset for the 1. TxPDO
		-------------------------------------------------------------------------------------------------------------------------------------------------------------	
		SyncTime 								USINT;			Cycle time of the sync telegram in ms. 
																Default = 0 : no sync will be started.
																If  SyncTime > 0, this FB initializes a sync telegram with the ID set at SyncCOBID. 
																The slave has to support synchronous communication 
		-------------------------------------------------------------------------------------------------------------------------------------------------------------
		SyncCOBID							UINT;			Index 1005h. ID of the sync telegram. Usually 16#80. IF 0, the ID won't be written.
		-------------------------------------------------------------------------------------------------------------------------------------------------------------
		SyncTimeOut 							INT := -1;		Index 1006h. Normally equal to SyncTime. 
																The slave usually set SyncTimeOut equal to SyncTime * 1.5. 
																If < 0, the index won't be written. 0 means no control over the sync interval 
		-------------------------------------------------------------------------------------------------------------------------------------------------------------
		stInitialParameter_COSlave 			MC_INITIALPARAMETER_COSLAVE;
												(*#################################################################
												With this struct, user defined parameters will be written to the BusCoupler after the
												initialization of the MPLC_ConnectUniversalSlave_CANopen. 
												Add the following code to your program to initialise the struct : 
												Example:
												Index 16#6423:	Activates the event-driven transmission of PDOs with analog inputs
												Index 16#3500:	Index from the manufacturer specific profile area
	
													stInitialParameter_COSlave.aIndex[1] := 16#6423;  	(* Index to write to *)
													stInitialParameter_COSlave.aSubIndex[1] := 0;   	(* SubIndex to write to *)
													stInitialParameter_COSlave.aBytes[1] := 1;   		(* Number of bytes to write  *)
													stInitialParameter_COSlave.aData[1] := 1;   			(* Data *)
	
													stInitialParameter_COSlave.aIndex[2] := 16#3500;  	(* Index to write to *)
													stInitialParameter_COSlave.aSubIndex[2] := 0;   	(* SubIndex to write to *)
													stInitialParameter_COSlave.aBytes[2] := 2;   		(* Number of bytes to write *)
													stInitialParameter_COSlave.aData[2] := 5;   			(* Data *)
	
												If there are more than 10 (DHP11B) or 64 (DHx41B) parameters to write, declare 
												NUMOF_INITIALPARAMETER in your program.
	
													VAR_GLOBAL CONSTANT
														NUMOF_INITIALPARAMETER : UDINT := 20;	
													END_VAR
	
												##################################################################*)

		bNoDeactivatePDO:			BOOL := FALSE; (* Change of Transmission Type, Inhibit- and Event- Time without deactivate RxPDO and TxPDO*)

			-------------------------------------------------------------------------------------------------------------------------------------------------------------
		(* IDs of the PDO telegrams. The IDs are always calculated with the following IDs as a basis + the address of the bus coupler *)

		RxPDO 								ARRAY[1..32] OF MC_PDO_COSLAVE;			(* MOVI-PLC --> Slave *)
												(* := 16#200,16#300,16#400,16#500,16#780,16#240,16#340,16#440,16#540,16#7C0;	*)
		-------------------------------------------------------------------------------------------------------------------------------------------------------------
		TxPDO 								ARRAY[1..32] OF MC_PDO_COSLAVE; 			(* Slave --> MOVI-PLC *)
												(*:= 16#180,16#280,16#380,16#480,16#680,16#1C0,16#2C0,16#3C0,16#4C0,16#6C0;*)
	*)
END_VAR
IF Enable AND NOT Done THEN

	(*########################################################

		Configuration of CANopenSlave HBM Waage)
		
		NOTE! 
		
	#########################################################

		TransmissionType for TxPDOs and RxPDOs:

			0:										Event controlled and sychron (with SYNC-Object)
			1-240:									Cyclic and synchron (with SYNC-Object)
			254:									Producer specified
			255:									Acyclic and eventcontrolled 
			255 and EventTime = InhibitTime:	Cyclic

	#########################################################	*)

	ExtConfig.bWaitBeforeOperational			:=FALSE;
	ExtConfig.bNoSettingsDownload				:=FALSE;
	ExtConfig.bResetUnconditional 				:=FALSE;
	ExtConfig.bIOHold							 :=FALSE;
	ExtConfig.TimeOutHeartBeat					 :=0;
	ExtConfig.bNoHeartBeat_Producer			 := FALSE; (*Index 1017 SubIndex 0 not available *)
	ExtConfig.TimeOutNodeGuarding			 :=100;
	ExtConfig.bNoNodeGuarding 				:= FALSE;(* the Index of NodeGuarding isn`t available *)
	ExtConfig.TimeOutInitSequence 				:=10;
	ExtConfig.SyncCOBID							:= 0;				(* SyncObject ID for TransmissionType 0-240 (RxPDO). Usually 128. If 0, the ID will not be written *)
	ExtConfig.SyncTime							:= 0;				(* CycleTime for the SYNC-Object *)



	(**************************************************** TxPDOs of CANOpenSlave ( MOVI-PLC ReceiveObjects) ************************************************************)

	ExtConfig.NumberOfTxPDO			:= 5;		(*  TxPDO ---> CANopenSlave Transmit *)
	ExtConfig.bNoTransmissionTyp_TxPDO := FALSE;(* Transmission Type for TxPDO not changeable *)
(* TxPDO ---> Sende-PDO1: Messwert/Status *)
	ExtConfig.TxPDO[1].EventTime		:= 0;		(* Master: CycleTime in ms for TransmitObjects (MOVI-PLC) *)
	ExtConfig.TxPDO[1].Length			:= 6;		(* Master: Length of this TransmitObject in bytes *)
	ExtConfig.TxPDO[1].TransmissionType := 254;
(*  TxPDO ---> Sende-PDO2: Triggerergebnis/Status *)
	ExtConfig.TxPDO[2].EventTime		:= 00;		(* Master: CycleTime in ms for TransmitObjects (MOVI-PLC) *)
	ExtConfig.TxPDO[2].Length			:= 6;		(* Master: Length of this TransmitObject in bytes *)
	ExtConfig.TxPDO[2].TransmissionType := 254;
(*  Sende PDO3: Dosierergebnis/Status  *)
	ExtConfig.TxPDO[3].EventTime		:= 00;		(* Master: CycleTime in ms for TransmitObjects (MOVI-PLC) *)
	ExtConfig.TxPDO[3].Length			:= 6;		(* Master: Length of this TransmitObject in bytes *)
	ExtConfig.TxPDO[3].TransmissionType := 254;
(*  TxPDO ---> Sende PDO4: Spitzenwerte Min und Max  *)
	ExtConfig.TxPDO[4].EventTime		:= 00;		(* Master: CycleTime in ms for TransmitObjects (MOVI-PLC) *)
	ExtConfig.TxPDO[4].Length			:= 8;		(* Master: Length of this TransmitObject in bytes *)
	ExtConfig.TxPDO[4].TransmissionType := 254;
(*  TxPDO ---> Sende-PDO5: Alarm Status *)
	ExtConfig.TxPDO[5].EventTime		:= 00;		(* Master: CycleTime in ms for TransmitObjects (MOVI-PLC) *)
	ExtConfig.TxPDO[5].Length			:= 4;	(* Master: Length of this TransmitObject in bytes *)
	ExtConfig.TxPDO[5].TransmissionType := 254;

	(*************************************************** RxPDOs of CANOpenSlave ( MOVI-PLC TransmitObjects) **********************************************************)

	ExtConfig.NumberOfRxPDO			:= 1;		(*  RxPDO ---> CANopenSlave Receive *)
	ExtConfig.bNoTransmissionTyp_RxPDO := FALSE;(* Transmission Type for RxPDO not changeable *)
	(* Empfangs-PDO: (Steuerwort)	^*)
	ExtConfig.RxPDO[1].InhibitTime		:= 0;		(* Master: InhibitTime in ms for TransmitObjects (MOVI-PLC) *)
	ExtConfig.RxPDO[1].Length			:= 2;		(* Master: Length of this TransmitObject in bytes *)
	ExtConfig.RxPDO[1].TransmissionType := 255;

	(***************************************************** Additional parameters to set in the CANOpenSlave  ***************************************************************)

	(* Set rotation direction *)
	ExtConfig.stInitialParameter_COSlave.aIndex[1]			:= 16#3400;
	ExtConfig.stInitialParameter_COSlave.aSubIndex[1]	:= 0;
	ExtConfig.stInitialParameter_COSlave.aBytes[1]		:= 4;
	ExtConfig.stInitialParameter_COSlave.aData[1]			:= 20;

	(********************************************** Additional configuration. Default values are in most cases sufficient *****************************************************)

	ExtConfig.bNoDeactivatePDO		 := TRUE; (* Change of Transmission Type, Inhibit- and Event- Time without deactivate RxPDO and TxPDO*)

	ExtConfig.TxPDO[1].COBID			:= 16#180;			(* Impossible to change*)
	ExtConfig.TxPDO[2].COBID			:= 16#280;			(* Impossible to change*)
	ExtConfig.TxPDO[3].COBID			:= 16#380;			 (* Impossible to change*)
	ExtConfig.TxPDO[4].COBID			:= 16#480;			(*480+	 Impossible to change*)
	ExtConfig.TxPDO[5].COBID			:= 16#1C0;			(* 300 + 3F Impossible to change*)

	ExtConfig.RxPDO[1].COBID			:= 16#200;		(* Impossible to change*)
	Done									 := TRUE;

END_IF
END_FUNCTION_BLOCK

(* POU CodeSamples/CANopen/UniversalMaster/FB_Configuration_CANopenSlave_LumbergCSL, ST *)
FUNCTION_BLOCK FB_Configuration_CANopenSlave_LumbergCSL
VAR_INPUT
	Enable: BOOL; 			(* Activate config *)
	Node: CAN_NODE;		(* Physical CAN where CAN module is connected:
										SBUS_NODE_1 := 1,
  										SBUS_NODE_2 := 2 *)
	Address: WORD; 			(* Address of the CANopen slave 1 - 63 *)
END_VAR
VAR_OUTPUT
	Done: BOOL;				(* Config done *)
END_VAR
VAR_IN_OUT
	ExtConfig : MC_EXTENDEDCONFIG_COSLAVE	;
	(*
		########################################################################################################
			MC_EXTENDEDCONFIG_COSLAVE
		#########################################################################################################

						
		Variable								Value			Description
		-------------------------------------------------------------------------------------------------------------------------------------------------------------
		bWaitBeforeOperational 				BOOL;			When TRUE, after the coupler has been parameterized, it won't be switched in operational
																before this variable is FALSE. This can be used for example, to store the configuration with the FB
																MPLC_Universal_CANopen, with Service "SEWIOS_STORE", after a reset of the coppler 
		-------------------------------------------------------------------------------------------------------------------------------------------------------------
		bNoSettingsDownload 				BOOL;			TRUE : No configuration of the module. The configuration has to be done manually.
		-------------------------------------------------------------------------------------------------------------------------------------------------------------
		bResetUnconditional 					BOOL;			Even if the Connect FB isn't in fault it is possible to reset the bus coppler
		-------------------------------------------------------------------------------------------------------------------------------------------------------------
		bIOHold 								BOOL;			TRUE : Input data remain unchanged and the output data are not resetet also if the FB is in fault 
		-------------------------------------------------------------------------------------------------------------------------------------------------------------
		TimeOutHeartBeat					UINT;			If this value (ms) is different to zero, HeartbeatMode will be activated
		-------------------------------------------------------------------------------------------------------------------------------------------------------------
		TimeOutNodeGuarding 				UINT;			If this value (ms) is different to zero, NodeGuarding will be activated. 
																Caution ! The MOVI-PLC basic doesn´t support NodeGuarding 
		-------------------------------------------------------------------------------------------------------------------------------------------------------------
		TimeOutInitSequence					UINT;			Timeout for initialisation sequence (seconds) 
		-------------------------------------------------------------------------------------------------------------------------------------------------------------
		NumberOfRxPDO 					UINT;			Receive PDO : MOVI-PLC --> Slave  max. 32 
		-------------------------------------------------------------------------------------------------------------------------------------------------------------
		NumberOfTxPDO 						UINT;			Send PDO :      Slave --> MOVI-PLC  max 32 
		-------------------------------------------------------------------------------------------------------------------------------------------------------------	
		SyncTime 								USINT;			Cycle time of the sync telegram in ms. 
																Default = 0 : no sync will be started.
																If  SyncTime > 0, this FB initializes a sync telegram with the ID set at SyncCOBID. 
																The slave has to support synchronous communication 
		-------------------------------------------------------------------------------------------------------------------------------------------------------------
		SyncCOBID							UINT;			Index 1005h. ID of the sync telegram. Usually 16#80. IF 0, the ID won't be written.
		-------------------------------------------------------------------------------------------------------------------------------------------------------------
		SyncTimeOut 							INT := -1;		Index 1006h. Normally equal to SyncTime. 
																The slave usually set SyncTimeOut equal to SyncTime * 1.5. 
																If < 0, the index won't be written. 0 means no control over the sync interval 
		-------------------------------------------------------------------------------------------------------------------------------------------------------------
		stInitialParameter_COSlave 			MC_INITIALPARAMETER_COSLAVE;
												(*#################################################################
												With this struct, user defined parameters will be written to the BusCoupler after the
												initialization of the MPLC_ConnectUniversalSlave_CANopen. 
												Add the following code to your program to initialise the struct : 
												Example:
												Index 16#6423:	Activates the event-driven transmission of PDOs with analog inputs
												Index 16#3500:	Index from the manufacturer specific profile area
	
													stInitialParameter_COSlave.aIndex[1] := 16#6423;  	(* Index to write to *)
													stInitialParameter_COSlave.aSubIndex[1] := 0;   	(* SubIndex to write to *)
													stInitialParameter_COSlave.aBytes[1] := 1;   		(* Number of bytes to write  *)
													stInitialParameter_COSlave.aData[1] := 1;   			(* Data *)
	
													stInitialParameter_COSlave.aIndex[2] := 16#3500;  	(* Index to write to *)
													stInitialParameter_COSlave.aSubIndex[2] := 0;   	(* SubIndex to write to *)
													stInitialParameter_COSlave.aBytes[2] := 2;   		(* Number of bytes to write *)
													stInitialParameter_COSlave.aData[2] := 5;   			(* Data *)
	
												If there are more than 10 (DHP11B) or 64 (DHx41B) parameters to write, declare 
												NUMOF_INITIALPARAMETER in your program.
	
													VAR_GLOBAL CONSTANT
														NUMOF_INITIALPARAMETER : UDINT := 20;	
													END_VAR
	
												##################################################################*)
			-------------------------------------------------------------------------------------------------------------------------------------------------------------
		(* IDs of the PDO telegrams. The IDs are always calculated with the following IDs as a basis + the address of the bus coupler *)

		RxPDO 								ARRAY[1..32] OF MC_PDO_COSLAVE;			(* MOVI-PLC --> Slave *)
												(* := 16#200,16#300,16#400,16#500,16#780,16#240,16#340,16#440,16#540,16#7C0;	*)
		-------------------------------------------------------------------------------------------------------------------------------------------------------------
		TxPDO 								ARRAY[1..32] OF MC_PDO_COSLAVE; 			(* Slave --> MOVI-PLC *)
												(*:= 16#180,16#280,16#380,16#480,16#680,16#1C0,16#2C0,16#3C0,16#4C0,16#6C0;*)
	*)
END_VAR

VAR
	bSend_SDO: BOOL;
	CanMsgSDO: ST_CanAcyclicMsg;
	parameterize: BOOL;
END_VAR
IF Enable AND NOT Done THEN

	(*########################################################

		Configuration of CANopenSlave (Lumberg 940 CSL 601)
		
	#########################################################*)

		IF NOT bSend_SDO THEN

		CanMsgSDO := F_WriteCanMsg(
							Node:=Node,
							ID:= 16#600 + Address,
							Length:= 8,
							Data1:= 16#2F01,
							Data2 := 16#3000,
							Data3 := 16#0200,
							Data4 := 0,
							SBUSGateway_LogAdr := 0 );
			IF CanMsgSDO.State = GEN_1_BUFFSTATE_INSERTED THEN
				bSend_SDO :=TRUE;
			END_IF
		ELSIF bSend_SDO THEN
			CanMsgSDO.Result := F_ResultCanMsg(CanAcyclicMsg:=CanMsgSDO);
			IF CanMsgSDO.Result = GEN_3_BUFFSTATE_COMPLETED_SUCCESSFUL THEN
				bSend_SDO:=FALSE;
				parameterize:=TRUE;
			ELSIF  CanMsgSDO.Result = GEN_5_BUFFSTATE_COMPLETED_MSG_LOST THEN
				(* Fehler beim Senden --> Nachricht ging verloren --> nochmals *)
				bSend_SDO :=FALSE;
			ELSIF  CanMsgSDO.Result = GEN_4_BUFFSTATE_COMPLETED_ERROR THEN
				(* Fehler beim Senden --> Non-recovery error from CAN --> nochmals *)
				bSend_SDO :=FALSE;
			END_IF
		END_IF

		P_AcyclicCommunicationTask_CAN;
	IF parameterize THEN

		(*#########################################################
	
			TransmissionType for TxPDOs and RxPDOs:
	
				0:										Event controlled and sychron (with SYNC-Object)
				1-240:									Cyclic and synchron (with SYNC-Object)
				254:									Producer specified
				255:									Acyclic and eventcontrolled 
				255 and EventTime = InhibitTime:	Cyclic
	
		#########################################################	*)
	
		ExtConfig.bNoDeactivatePDO		 := TRUE; (* Change of Transmission Type, Inhibit- and Event- Time without deactivate RxPDO and TxPDO*)
		(*************************************************** TxPDOs of CANOpenSlave ( MOVI-PLC ReceiveObjects) ***********************************************************)
	
		ExtConfig.NumberOfTxPDO				:= 1;		(*  TxPDO ---> CANopenSlave Transmit *)
	
		ExtConfig.TxPDO[1].EventTime			:= 100;		(* Slave: Index 0x18xx SubIndex 5: CycleTime in ms for CANopenSlave TXPDO *)
		ExtConfig.TxPDO[1].InhibitTime			:= 5;		(* Slave: Index 0x18xx SubIndex 3: InhibitTime in ms for CANopenSlave TxPDO *)
		ExtConfig.TxPDO[1].TransmissionType	:= 255;		(* Slave: Index 0x18xx SubIndex 2: TransmissionType for this TxPDO *)
	(*
		ExtConfig.TxPDO[2].EventTime			:= 100;		(* Slave: Index 0x18xx SubIndex 5: CycleTime in ms for CANopenSlave TXPDO *)
		ExtConfig.TxPDO[2].InhibitTime			:= 5;		(* Slave: Index 0x18xx SubIndex 3: InhibitTime in ms for CANopenSlave TxPDO *)
		ExtConfig.TxPDO[2].TransmissionType	:= 255;		(* Slave: Index 0x18xx SubIndex 2: TransmissionType for this TxPDO *)
	
		ExtConfig.TxPDO[3].EventTime			:= 100;		(* Slave: Index 0x18xx SubIndex 5: CycleTime in ms for CANopenSlave TXPDO *)
		ExtConfig.TxPDO[3].InhibitTime			:= 5;		(* Slave: Index 0x18xx SubIndex 3: InhibitTime in ms for CANopenSlave TxPDO *)
		ExtConfig.TxPDO[3].TransmissionType	:= 255;		(* Slave: Index 0x18xx SubIndex 2: TransmissionType for this TxPDO *)
	
		ExtConfig.TxPDO[4].EventTime			:= 100;		(* Slave: Index 0x18xx SubIndex 5: CycleTime in ms for CANopenSlave TXPDO *)
		ExtConfig.TxPDO[4].InhibitTime			:= 5;		(* Slave: Index 0x18xx SubIndex 3: InhibitTime in ms for CANopenSlave TxPDO *)
		ExtConfig.TxPDO[4].TransmissionType	:= 255;		(* Slave: Index 0x18xx SubIndex 2: TransmissionType for this TxPDO *)
	*)
	
		(*************************************************** RxPDOs of CANOpenSlave ( MOVI-PLC TransmitObjects) **********************************************************)
	
		ExtConfig.NumberOfRxPDO				:= 1;		(*  RxPDO ---> CANopenSlave Receive *)
	
		ExtConfig.RxPDO[1].EventTime			:= 100;		(* Master: CycleTime in ms for TransmitObjects (MOVI-PLC) *)
		ExtConfig.RxPDO[1].InhibitTime			:= 5;		(* Master: InhibitTime in ms for TransmitObjects (MOVI-PLC) *)
		ExtConfig.RxPDO[1].Length				:= 8;		(* Master: Length of this TransmitObject in bytes *)
		ExtConfig.RxPDO[1].TransmissionType	:= 255;		(* Slave: Index 0x14xx SubIndex 2: TransmissionType for this RxPDO *)
	(*
		ExtConfig.RxPDO[2].EventTime			:= 100;		(* Master: CycleTime in ms for TransmitObjects (MOVI-PLC) *)
		ExtConfig.RxPDO[2].InhibitTime			:= 5;		(* Master: InhibitTime in ms for TransmitObjects (MOVI-PLC) *)
		ExtConfig.RxPDO[2].Length				:= 8;		(* Master: Length of this TransmitObject in bytes *)
		ExtConfig.RxPDO[2].TransmissionType	:= 255;		(* Slave: Index 0x14xx SubIndex 2: TransmissionType for this RxPDO *)
	
		ExtConfig.RxPDO[3].EventTime			:= 100;		(* Master: CycleTime in ms for TransmitObjects (MOVI-PLC) *)
		ExtConfig.RxPDO[3].InhibitTime			:= 5;		(* Master: InhibitTime in ms for TransmitObjects (MOVI-PLC) *)
		ExtConfig.RxPDO[3].Length				:= 8;		(* Master: Length of this TransmitObject in bytes *)
		ExtConfig.RxPDO[3].TransmissionType	:= 255;		(* Slave: Index 0x14xx SubIndex 2: TransmissionType for this RxPDO *)
	
		ExtConfig.RxPDO[4].EventTime			:= 100;		(* Master: CycleTime in ms for TransmitObjects (MOVI-PLC) *)
		ExtConfig.RxPDO[4].InhibitTime			:= 5;		(* Master: InhibitTime in ms for TransmitObjects (MOVI-PLC) *)
		ExtConfig.RxPDO[4].Length				:= 8;		(* Master: Length of this TransmitObject in bytes *)
		ExtConfig.RxPDO[4].TransmissionType	:= 255;		(* Slave: Index 0x14xx SubIndex 2: TransmissionType for this RxPDO *)
	*)
	
		(***************************************************** Additional parameters to set in the CANOpenSlave  ***************************************************************)
	
	(*	(* Enable transmission of analog inputs *)
		ExtConfig.stInitialParameter_COSlave.aIndex[1]			:= 16#6423;
		ExtConfig.stInitialParameter_COSlave.aSubIndex[1]	:= 0;
		ExtConfig.stInitialParameter_COSlave.aBytes[1]		:= 1;
		ExtConfig.stInitialParameter_COSlave.aData[1]			:= 1;*)
		(* Enable transmission of analog inputs *)
	
	
		(********************************************** Additional configuration. Default values are in most cases sufficient *****************************************************)
	
		ExtConfig.bIOHold						:= FALSE;
		ExtConfig.bNoSettingsDownload			:= FALSE;
		ExtConfig.bWaitBeforeOperational		:= FALSE;
		ExtConfig.bResetUnconditional			:= FALSE;
	
		ExtConfig.TimeOutHeartBeat				:= 400;				(* [ms] *)
		ExtConfig.TimeOutNodeGuarding		:= 0;				(* [ms]. CAUTION ! DHP11B (MOVI-PLC basic) does NOT support NodeGuarding *)
		ExtConfig.TimeOutInitSequence			:= 10;				(* [seconds]. If the Init-Sequence takes longer than this TimeOut time --> Error *)
		ExtConfig.SyncCOBID						:= 0;				(* SyncObject ID for TransmissionType 0-240 (RxPDO). Usually 128. If 0, the ID will not be written *)
		ExtConfig.SyncTime						:= 0;				(* CycleTime for the SYNC-Object *)
	
		ExtConfig.TxPDO[1].COBID				:= 16#180;			(* In order to disable the use of RTR frames for the PDOs, set bit 30 = "RTR not allowed" *)
		ExtConfig.TxPDO[2].COBID				:= 16#280;			(* Ex. 16#4000_0280 *)
		ExtConfig.TxPDO[3].COBID				:= 16#380;
		ExtConfig.TxPDO[4].COBID				:= 16#480;			(* NOTE! These values are base values. The input "Address" will automatically be added *)
		ExtConfig.TxPDO[5].COBID				:= 16#680;
		ExtConfig.TxPDO[6].COBID				:= 16#1C0;
		ExtConfig.TxPDO[7].COBID				:= 16#2C0;
		ExtConfig.TxPDO[8].COBID				:= 16#3C0;
		ExtConfig.TxPDO[9].COBID				:= 16#4C0;
		ExtConfig.TxPDO[10].COBID				:= 16#6C0;
	
		ExtConfig.RxPDO[1].COBID				:= 16#200;
		ExtConfig.RxPDO[2].COBID				:= 16#300;
		ExtConfig.RxPDO[3].COBID				:= 16#400;
		ExtConfig.RxPDO[4].COBID				:= 16#500;
		ExtConfig.RxPDO[5].COBID				:= 16#780;
		ExtConfig.RxPDO[6].COBID				:= 16#240;
		ExtConfig.RxPDO[7].COBID				:= 16#340;
		ExtConfig.RxPDO[8].COBID				:= 16#440;
		ExtConfig.RxPDO[9].COBID				:= 16#540;
		ExtConfig.RxPDO[10].COBID				:= 16#7C0;
	
	
	
		Done := TRUE;
		parameterize := FALSE;
	END_IF
END_IF
END_FUNCTION_BLOCK

(* POU CodeSamples/CANopen/UniversalMaster/FB_Configuration_CANopenSlave_MURRCUBE67, ST *)
FUNCTION_BLOCK FB_Configuration_CANopenSlave_MURRCUBE67
VAR_INPUT
	Enable: BOOL; 			(* Activate config *)
END_VAR
VAR_OUTPUT
	Done: BOOL;				(* Config done *)
END_VAR
VAR_IN_OUT
	ExtConfig : MC_EXTENDEDCONFIG_COSLAVE	;
	(*
		########################################################################################################
			MC_EXTENDEDCONFIG_COSLAVE
		#########################################################################################################

						
		Variable								Value			Description
		-------------------------------------------------------------------------------------------------------------------------------------------------------------
		bWaitBeforeOperational 				BOOL;			When TRUE, after the coupler has been parameterized, it won't be switched in operational
																before this variable is FALSE. This can be used for example, to store the configuration with the FB
																MPLC_Universal_CANopen, with Service "SEWIOS_STORE", after a reset of the coppler 
		-------------------------------------------------------------------------------------------------------------------------------------------------------------
		bNoSettingsDownload 				BOOL;			TRUE : No configuration of the module. The configuration has to be done manually.
		-------------------------------------------------------------------------------------------------------------------------------------------------------------
		bResetUnconditional 					BOOL;			Even if the Connect FB isn't in fault it is possible to reset the bus coppler
		-------------------------------------------------------------------------------------------------------------------------------------------------------------
		bIOHold 								BOOL;			TRUE : Input data remain unchanged and the output data are not resetet also if the FB is in fault 
		-------------------------------------------------------------------------------------------------------------------------------------------------------------
		TimeOutHeartBeat					UINT;			If this value (ms) is different to zero, HeartbeatMode will be activated
		-------------------------------------------------------------------------------------------------------------------------------------------------------------
		TimeOutNodeGuarding 				UINT;			If this value (ms) is different to zero, NodeGuarding will be activated. 
																Caution ! The MOVI-PLC basic doesn´t support NodeGuarding 
		-------------------------------------------------------------------------------------------------------------------------------------------------------------
		TimeOutInitSequence					UINT;			Timeout for initialisation sequence (seconds) 
		-------------------------------------------------------------------------------------------------------------------------------------------------------------
		NumberOfRxPDO 					UINT;			Receive PDO : MOVI-PLC --> Slave  max. 32 
		-------------------------------------------------------------------------------------------------------------------------------------------------------------
		NumberOfTxPDO 						UINT;			Send PDO :      Slave --> MOVI-PLC  max 32 
		-------------------------------------------------------------------------------------------------------------------------------------------------------------	
		SyncTime 								USINT;			Cycle time of the sync telegram in ms. 
																Default = 0 : no sync will be started.
																If  SyncTime > 0, this FB initializes a sync telegram with the ID set at SyncCOBID. 
																The slave has to support synchronous communication 
		-------------------------------------------------------------------------------------------------------------------------------------------------------------
		SyncCOBID							UINT;			Index 1005h. ID of the sync telegram. Usually 16#80. IF 0, the ID won't be written.
		-------------------------------------------------------------------------------------------------------------------------------------------------------------
		SyncTimeOut 							INT := -1;		Index 1006h. Normally equal to SyncTime. 
																The slave usually set SyncTimeOut equal to SyncTime * 1.5. 
																If < 0, the index won't be written. 0 means no control over the sync interval 
		-------------------------------------------------------------------------------------------------------------------------------------------------------------
		stInitialParameter_COSlave 			MC_INITIALPARAMETER_COSLAVE;
												(*#################################################################
												With this struct, user defined parameters will be written to the BusCoupler after the
												initialization of the MPLC_ConnectUniversalSlave_CANopen. 
												Add the following code to your program to initialise the struct : 
												Example:
												Index 16#6423:	Activates the event-driven transmission of PDOs with analog inputs
												Index 16#3500:	Index from the manufacturer specific profile area
	
													stInitialParameter_COSlave.aIndex[1] := 16#6423;  	(* Index to write to *)
													stInitialParameter_COSlave.aSubIndex[1] := 0;   	(* SubIndex to write to *)
													stInitialParameter_COSlave.aBytes[1] := 1;   		(* Number of bytes to write  *)
													stInitialParameter_COSlave.aData[1] := 1;   			(* Data *)
	
													stInitialParameter_COSlave.aIndex[2] := 16#3500;  	(* Index to write to *)
													stInitialParameter_COSlave.aSubIndex[2] := 0;   	(* SubIndex to write to *)
													stInitialParameter_COSlave.aBytes[2] := 2;   		(* Number of bytes to write *)
													stInitialParameter_COSlave.aData[2] := 5;   			(* Data *)
	
												If there are more than 10 (DHP11B) or 64 (DHx41B) parameters to write, declare 
												NUMOF_INITIALPARAMETER in your program.
	
													VAR_GLOBAL CONSTANT
														NUMOF_INITIALPARAMETER : UDINT := 20;	
													END_VAR
	
												##################################################################*)
			-------------------------------------------------------------------------------------------------------------------------------------------------------------
		(* IDs of the PDO telegrams. The IDs are always calculated with the following IDs as a basis + the address of the bus coupler *)

		RxPDO 								ARRAY[1..32] OF MC_PDO_COSLAVE;			(* MOVI-PLC --> Slave *)
												(* := 16#200,16#300,16#400,16#500,16#780,16#240,16#340,16#440,16#540,16#7C0;	*)
		-------------------------------------------------------------------------------------------------------------------------------------------------------------
		TxPDO 								ARRAY[1..32] OF MC_PDO_COSLAVE; 			(* Slave --> MOVI-PLC *)
												(*:= 16#180,16#280,16#380,16#480,16#680,16#1C0,16#2C0,16#3C0,16#4C0,16#6C0;*)
	*)
END_VAR
IF Enable AND NOT Done THEN

	(*########################################################

		Configuration of CANopenSlave MURR CUBE67
		
